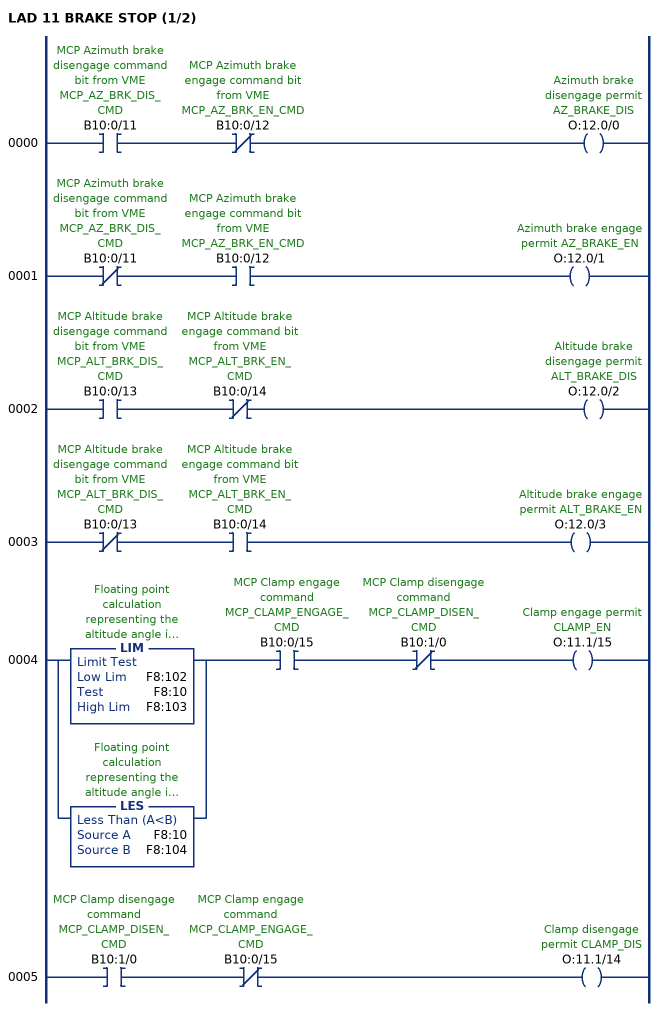
% Rung: 0 %
SOR XIC B10:0/11 XIO B10:0/12 OTE O:12.0/0 EOR
%   B10:0/11  MCP_AZ_BRK_DIS_CMD  "MCP Azimuth brake disengage command bit from VME" %
%   B10:0/12  MCP_AZ_BRK_EN_CMD  "MCP Azimuth brake engage command bit from VME" %
%   O:12.0/0  AZ_BRAKE_DIS  "Azimuth brake disengage permit" %
% Rung: 1 %
SOR XIO B10:0/11 XIC B10:0/12 OTE O:12.0/1 EOR
%   B10:0/11  MCP_AZ_BRK_DIS_CMD  "MCP Azimuth brake disengage command bit from VME" %
%   B10:0/12  MCP_AZ_BRK_EN_CMD  "MCP Azimuth brake engage command bit from VME" %
%   O:12.0/1  AZ_BRAKE_EN  "Azimuth brake engage permit" %
% Rung: 2 %
SOR XIC B10:0/13 XIO B10:0/14 OTE O:12.0/2 EOR
%   B10:0/13  MCP_ALT_BRK_DIS_CMD  "MCP Altitude brake disengage command bit from VME" %
%   B10:0/14  MCP_ALT_BRK_EN_CMD  "MCP Altitude brake engage command bit from VME" %
%   O:12.0/2  ALT_BRAKE_DIS  "Altitude brake disengage permit" %
% Rung: 3 %
SOR XIO B10:0/13 XIC B10:0/14 OTE O:12.0/3 EOR
%   B10:0/13  MCP_ALT_BRK_DIS_CMD  "MCP Altitude brake disengage command bit from VME" %
%   B10:0/14  MCP_ALT_BRK_EN_CMD  "MCP Altitude brake engage command bit from VME" %
%   O:12.0/3  ALT_BRAKE_EN  "Altitude brake engage permit" %
% Rung: 4 %
SOR BST LIM F8:102 F8:10 F8:103 NXB LES F8:10 F8:104 BND XIC B10:0/15 XIO B10:1/0 OTE O:11.1/15 EOR
%   F8:102  CLAMP_LOW_LIMIT  "The azimuth clamp will work above this limit and below CLAMP_HIGH_LIMIT" %
%   F8:10  ALT_ANGLE  "Floating point calculation representing the altitude angle in degrees." %
%   F8:103  CLAMP_HIGH_LIMIT  "The azimuth clamp will work below this limit and above CLAMP_LOW_LIMIT" %
%   F8:104  CLAMP_STOW_LIMIT  "The azimuth clamp will work below this limit" %
%   B10:0/15  MCP_CLAMP_ENGAGE_CMD  "MCP Clamp engage command" %
%   B10:1/0  MCP_CLAMP_DISEN_CMD  "MCP Clamp disengage command" %
%   O:11.1/15  CLAMP_EN  "Clamp engage permit" %
% Rung: 5 %
SOR XIC B10:1/0 XIO B10:0/15 OTE O:11.1/14 EOR
%   B10:1/0  MCP_CLAMP_DISEN_CMD  "MCP Clamp disengage command" %
%   B10:0/15  MCP_CLAMP_ENGAGE_CMD  "MCP Clamp engage command" %
%   O:11.1/14  CLAMP_DIS  "Clamp disengage permit" %

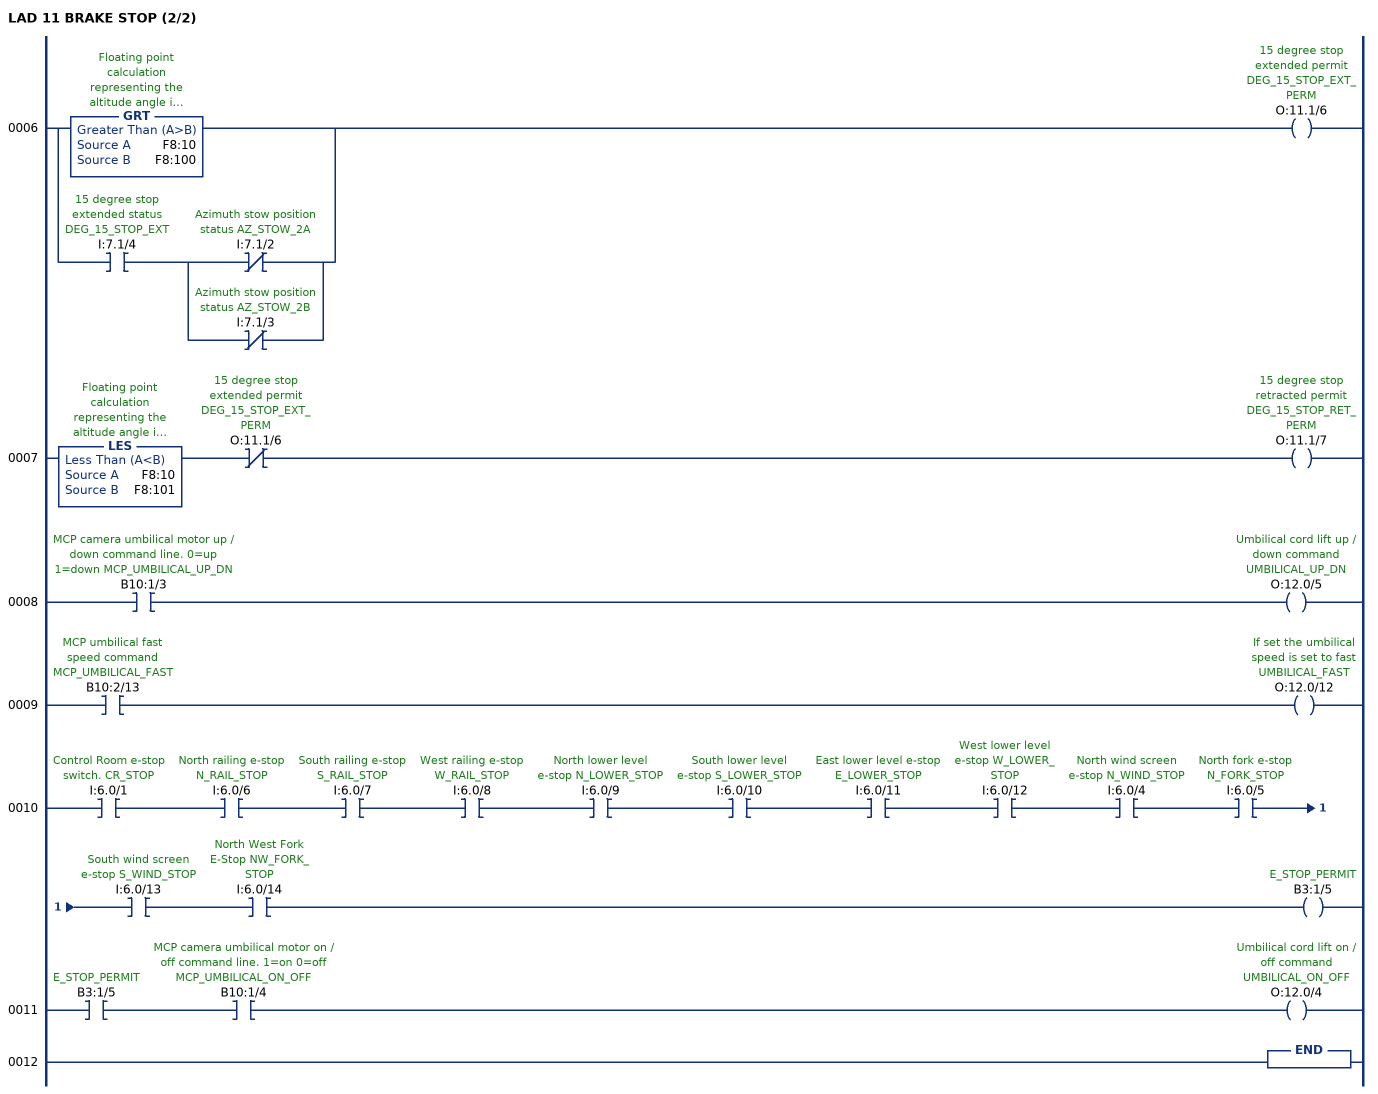
% Rung: 6 %
SOR BST GRT F8:10 F8:100 NXB XIC I:7.1/4 BST XIO I:7.1/2 NXB XIO I:7.1/3 BND BND OTE O:11.1/6 EOR
%   F8:10  ALT_ANGLE  "Floating point calculation representing the altitude angle in degrees." %
%   F8:100  DEG_15_STOP_EXT_LMT  "The 15 Degree stop extends at this value" %
%   I:7.1/4  DEG_15_STOP_EXT  "15 degree stop extended status" %
%   I:7.1/2  AZ_STOW_2A  "Azimuth stow position status" %
%   I:7.1/3  AZ_STOW_2B  "Azimuth stow position status" %
%   O:11.1/6  DEG_15_STOP_EXT_PERM  "15 degree stop extended permit" %
% Rung: 7 %
SOR LES F8:10 F8:101 XIO O:11.1/6 OTE O:11.1/7 EOR
%   F8:10  ALT_ANGLE  "Floating point calculation representing the altitude angle in degrees." %
%   F8:101  DEG_15_STOP_RET_LMT  "The 15 Degree stop retracts at this value" %
%   O:11.1/6  DEG_15_STOP_EXT_PERM  "15 degree stop extended permit" %
%   O:11.1/7  DEG_15_STOP_RET_PERM  "15 degree stop retracted permit" %
% Rung: 8 %
SOR XIC B10:1/3 OTE O:12.0/5 EOR
%   B10:1/3  MCP_UMBILICAL_UP_DN  "MCP camera umbilical motor up / down command line. 0=up 1=down" %
%   O:12.0/5  UMBILICAL_UP_DN  "Umbilical cord lift up / down command" %
% Rung: 9 %
SOR XIC B10:2/13 OTE O:12.0/12 EOR
%   B10:2/13  MCP_UMBILICAL_FAST  "MCP umbilical fast speed command" %
%   O:12.0/12  UMBILICAL_FAST  "If set the umbilical speed is set to fast" %
% Rung: 10 %
SOR XIC I:6.0/1 XIC I:6.0/6 XIC I:6.0/7 XIC I:6.0/8 XIC I:6.0/9 XIC I:6.0/10 XIC I:6.0/11 XIC I:6.0/12 XIC I:6.0/4 XIC I:6.0/5 XIC I:6.0/13 XIC I:6.0/14 OTE B3:1/5 EOR
%   I:6.0/1  CR_STOP  "Control Room e-stop switch." %
%   I:6.0/6  N_RAIL_STOP  "North railing e-stop" %
%   I:6.0/7  S_RAIL_STOP  "South railing e-stop" %
%   I:6.0/8  W_RAIL_STOP  "West railing e-stop" %
%   I:6.0/9  N_LOWER_STOP  "North lower level e-stop" %
%   I:6.0/10  S_LOWER_STOP  "South lower level e-stop" %
%   I:6.0/11  E_LOWER_STOP  "East lower level e-stop" %
%   I:6.0/12  W_LOWER_STOP  "West lower level e-stop" %
%   I:6.0/4  N_WIND_STOP  "North wind screen e-stop" %
%   I:6.0/5  N_FORK_STOP  "North fork e-stop" %
%   I:6.0/13  S_WIND_STOP  "South wind screen e-stop" %
%   I:6.0/14  NW_FORK_STOP  "North West Fork E-Stop" %
%   B3:1/5  E_STOP_PERMIT %
% Rung: 11 %
SOR XIC B3:1/5 XIC B10:1/4 OTE O:12.0/4 EOR
%   B3:1/5  E_STOP_PERMIT %
%   B10:1/4  MCP_UMBILICAL_ON_OFF  "MCP camera umbilical motor on / off command line. 1=on 0=off" %
%   O:12.0/4  UMBILICAL_ON_OFF  "Umbilical cord lift on / off command" %
% Rung: 12 %
SOR END EOR

LADDER 12 "E-STOP SW"
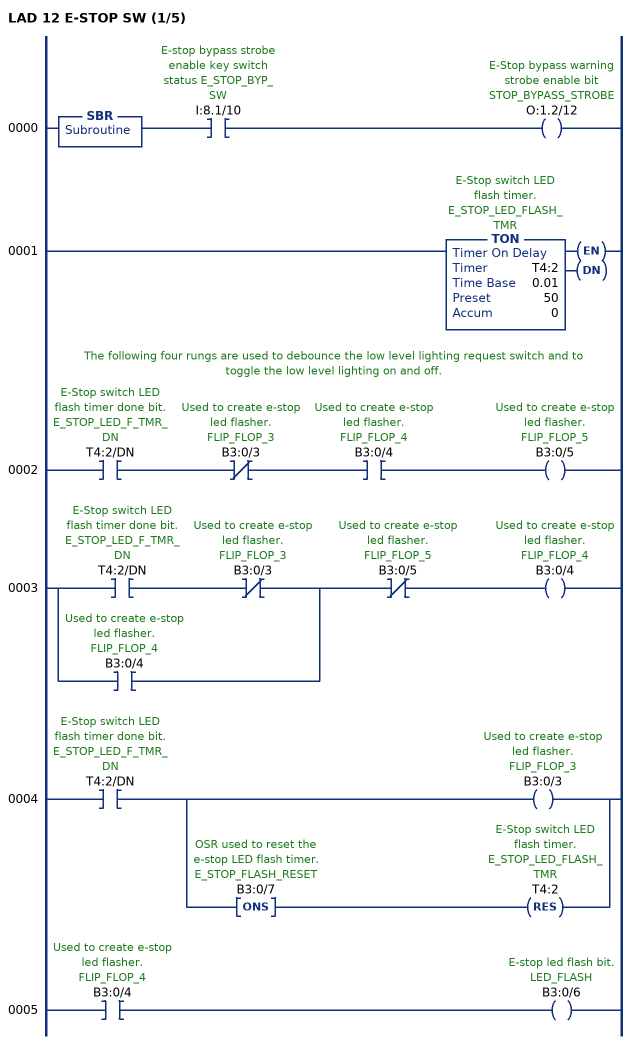
% Rung: 0 %
SOR SBR XIC I:8.1/10 OTE O:1.2/12 EOR
%   I:8.1/10  E_STOP_BYP_SW  "E-stop bypass strobe enable key switch status" %
%   O:1.2/12  STOP_BYPASS_STROBE  "E-Stop bypass warning strobe enable bit" %
% Rung: 1 %
SOR TON T4:2 0.01 50 0 EOR
%   T4:2  E_STOP_LED_FLASH_TMR  "E-Stop switch LED flash timer." %
% Rung: 2 %
% The following four rungs are used to debounce the low level lighting request switch and to toggle the low level lighting on and off. %
SOR XIC T4:2/DN XIO B3:0/3 XIC B3:0/4 OTE B3:0/5 EOR
%   T4:2/DN  E_STOP_LED_F_TMR_DN  "E-Stop switch LED flash timer done bit." %
%   B3:0/3  FLIP_FLOP_3  "Used to create e-stop led flasher." %
%   B3:0/4  FLIP_FLOP_4  "Used to create e-stop led flasher." %
%   B3:0/5  FLIP_FLOP_5  "Used to create e-stop led flasher." %
% Rung: 3 %
SOR BST XIC T4:2/DN XIO B3:0/3 NXB XIC B3:0/4 BND XIO B3:0/5 OTE B3:0/4 EOR
%   T4:2/DN  E_STOP_LED_F_TMR_DN  "E-Stop switch LED flash timer done bit." %
%   B3:0/3  FLIP_FLOP_3  "Used to create e-stop led flasher." %
%   B3:0/4  FLIP_FLOP_4  "Used to create e-stop led flasher." %
%   B3:0/5  FLIP_FLOP_5  "Used to create e-stop led flasher." %
% Rung: 4 %
SOR XIC T4:2/DN BST OTE B3:0/3 NXB OSR B3:0/7 RES T4:2 BND EOR
%   T4:2/DN  E_STOP_LED_F_TMR_DN  "E-Stop switch LED flash timer done bit." %
%   B3:0/3  FLIP_FLOP_3  "Used to create e-stop led flasher." %
%   B3:0/7  E_STOP_FLASH_RESET  "OSR used to reset the e-stop LED flash timer." %
%   T4:2  E_STOP_LED_FLASH_TMR  "E-Stop switch LED flash timer." %
% Rung: 5 %
SOR XIC B3:0/4 OTE B3:0/6 EOR
%   B3:0/4  FLIP_FLOP_4  "Used to create e-stop led flasher." %
%   B3:0/6  LED_FLASH  "E-stop led flash bit." %

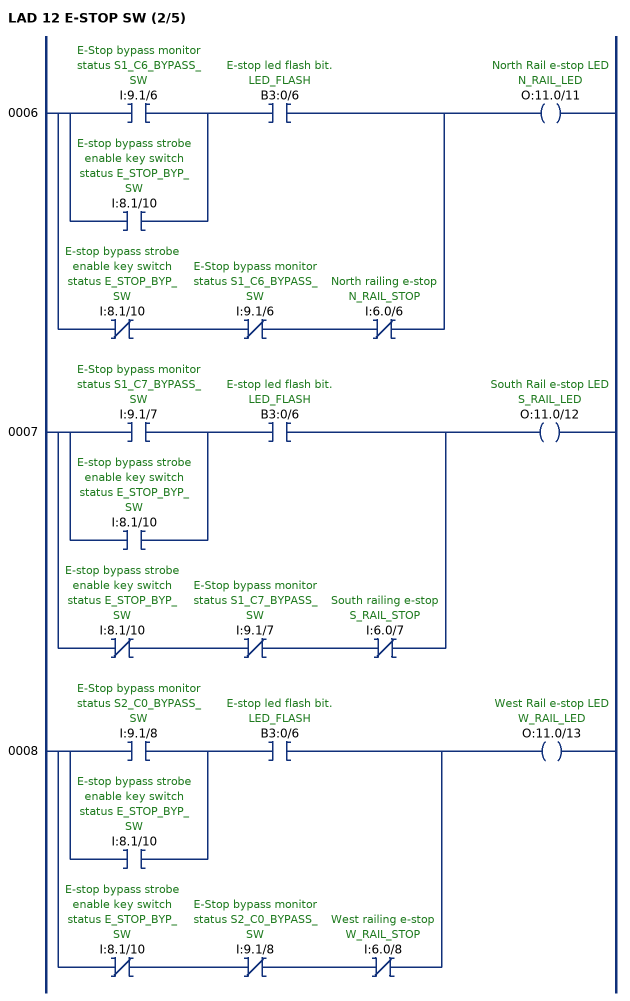
% Rung: 6 %
SOR BST BST XIC I:9.1/6 NXB XIC I:8.1/10 BND XIC B3:0/6 NXB XIO I:8.1/10 XIO I:9.1/6 XIO I:6.0/6 BND OTE O:11.0/11 EOR
%   I:9.1/6  S1_C6_BYPASS_SW  "E-Stop bypass monitor status" %
%   I:8.1/10  E_STOP_BYP_SW  "E-stop bypass strobe enable key switch status" %
%   B3:0/6  LED_FLASH  "E-stop led flash bit." %
%   I:6.0/6  N_RAIL_STOP  "North railing e-stop" %
%   O:11.0/11  N_RAIL_LED  "North Rail e-stop LED" %
% Rung: 7 %
SOR BST BST XIC I:9.1/7 NXB XIC I:8.1/10 BND XIC B3:0/6 NXB XIO I:8.1/10 XIO I:9.1/7 XIO I:6.0/7 BND OTE O:11.0/12 EOR
%   I:9.1/7  S1_C7_BYPASS_SW  "E-Stop bypass monitor status" %
%   I:8.1/10  E_STOP_BYP_SW  "E-stop bypass strobe enable key switch status" %
%   B3:0/6  LED_FLASH  "E-stop led flash bit." %
%   I:6.0/7  S_RAIL_STOP  "South railing e-stop" %
%   O:11.0/12  S_RAIL_LED  "South Rail e-stop LED" %
% Rung: 8 %
SOR BST BST XIC I:9.1/8 NXB XIC I:8.1/10 BND XIC B3:0/6 NXB XIO I:8.1/10 XIO I:9.1/8 XIO I:6.0/8 BND OTE O:11.0/13 EOR
%   I:9.1/8  S2_C0_BYPASS_SW  "E-Stop bypass monitor status" %
%   I:8.1/10  E_STOP_BYP_SW  "E-stop bypass strobe enable key switch status" %
%   B3:0/6  LED_FLASH  "E-stop led flash bit." %
%   I:6.0/8  W_RAIL_STOP  "West railing e-stop" %
%   O:11.0/13  W_RAIL_LED  "West Rail e-stop LED" %

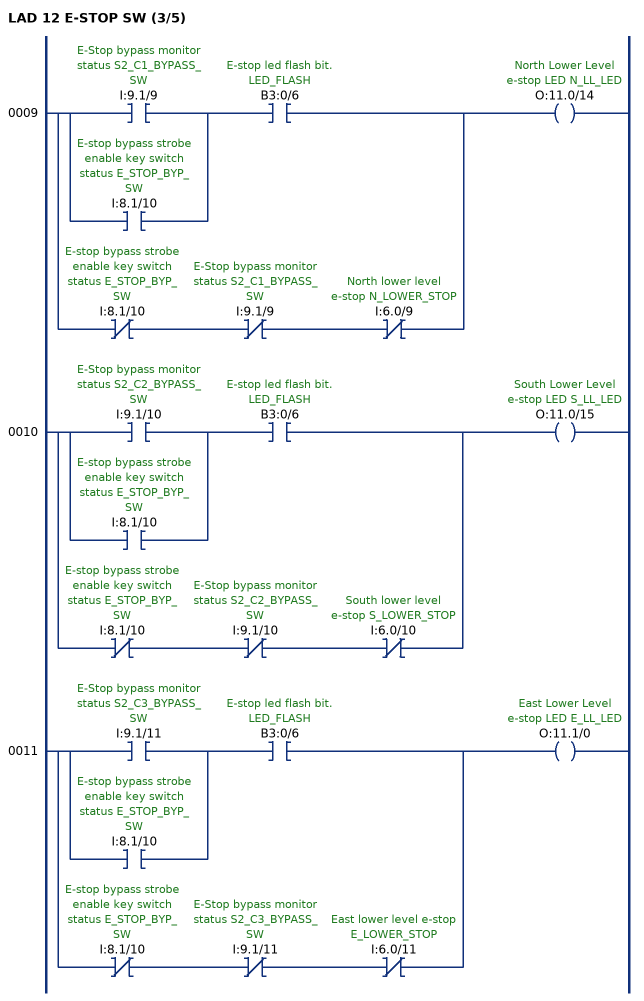
% Rung: 9 %
SOR BST BST XIC I:9.1/9 NXB XIC I:8.1/10 BND XIC B3:0/6 NXB XIO I:8.1/10 XIO I:9.1/9 XIO I:6.0/9 BND OTE O:11.0/14 EOR
%   I:9.1/9  S2_C1_BYPASS_SW  "E-Stop bypass monitor status" %
%   I:8.1/10  E_STOP_BYP_SW  "E-stop bypass strobe enable key switch status" %
%   B3:0/6  LED_FLASH  "E-stop led flash bit." %
%   I:6.0/9  N_LOWER_STOP  "North lower level e-stop" %
%   O:11.0/14  N_LL_LED  "North Lower Level e-stop LED" %
% Rung: 10 %
SOR BST BST XIC I:9.1/10 NXB XIC I:8.1/10 BND XIC B3:0/6 NXB XIO I:8.1/10 XIO I:9.1/10 XIO I:6.0/10 BND OTE O:11.0/15 EOR
%   I:9.1/10  S2_C2_BYPASS_SW  "E-Stop bypass monitor status" %
%   I:8.1/10  E_STOP_BYP_SW  "E-stop bypass strobe enable key switch status" %
%   B3:0/6  LED_FLASH  "E-stop led flash bit." %
%   I:6.0/10  S_LOWER_STOP  "South lower level e-stop" %
%   O:11.0/15  S_LL_LED  "South Lower Level e-stop LED" %
% Rung: 11 %
SOR BST BST XIC I:9.1/11 NXB XIC I:8.1/10 BND XIC B3:0/6 NXB XIO I:8.1/10 XIO I:9.1/11 XIO I:6.0/11 BND OTE O:11.1/0 EOR
%   I:9.1/11  S2_C3_BYPASS_SW  "E-Stop bypass monitor status" %
%   I:8.1/10  E_STOP_BYP_SW  "E-stop bypass strobe enable key switch status" %
%   B3:0/6  LED_FLASH  "E-stop led flash bit." %
%   I:6.0/11  E_LOWER_STOP  "East lower level e-stop" %
%   O:11.1/0  E_LL_LED  "East Lower Level e-stop LED" %

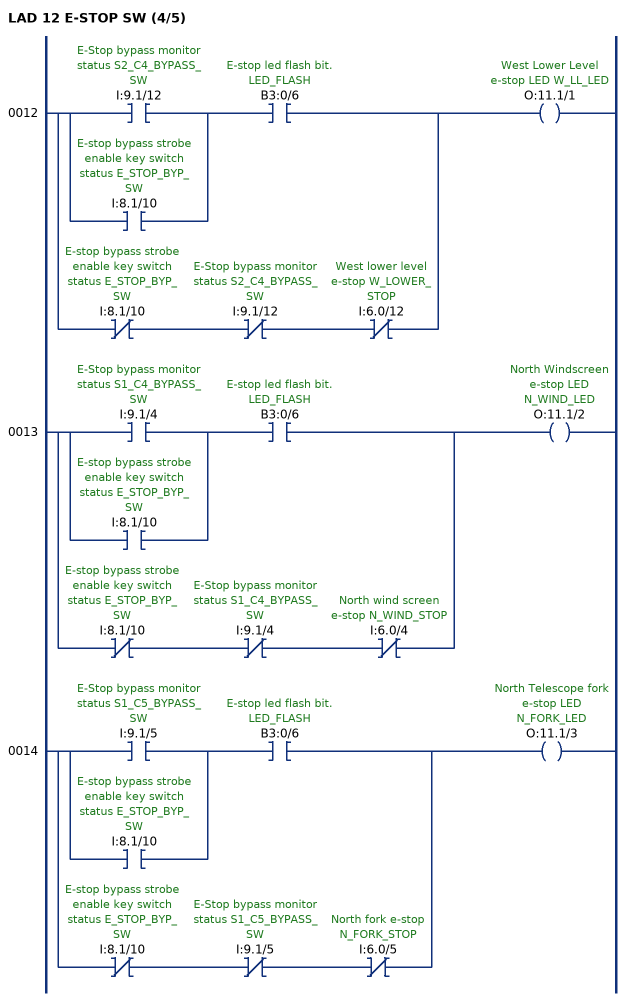
% Rung: 12 %
SOR BST BST XIC I:9.1/12 NXB XIC I:8.1/10 BND XIC B3:0/6 NXB XIO I:8.1/10 XIO I:9.1/12 XIO I:6.0/12 BND OTE O:11.1/1 EOR
%   I:9.1/12  S2_C4_BYPASS_SW  "E-Stop bypass monitor status" %
%   I:8.1/10  E_STOP_BYP_SW  "E-stop bypass strobe enable key switch status" %
%   B3:0/6  LED_FLASH  "E-stop led flash bit." %
%   I:6.0/12  W_LOWER_STOP  "West lower level e-stop" %
%   O:11.1/1  W_LL_LED  "West Lower Level e-stop LED" %
% Rung: 13 %
SOR BST BST XIC I:9.1/4 NXB XIC I:8.1/10 BND XIC B3:0/6 NXB XIO I:8.1/10 XIO I:9.1/4 XIO I:6.0/4 BND OTE O:11.1/2 EOR
%   I:9.1/4  S1_C4_BYPASS_SW  "E-Stop bypass monitor status" %
%   I:8.1/10  E_STOP_BYP_SW  "E-stop bypass strobe enable key switch status" %
%   B3:0/6  LED_FLASH  "E-stop led flash bit." %
%   I:6.0/4  N_WIND_STOP  "North wind screen e-stop" %
%   O:11.1/2  N_WIND_LED  "North Windscreen e-stop LED" %
% Rung: 14 %
SOR BST BST XIC I:9.1/5 NXB XIC I:8.1/10 BND XIC B3:0/6 NXB XIO I:8.1/10 XIO I:9.1/5 XIO I:6.0/5 BND OTE O:11.1/3 EOR
%   I:9.1/5  S1_C5_BYPASS_SW  "E-Stop bypass monitor status" %
%   I:8.1/10  E_STOP_BYP_SW  "E-stop bypass strobe enable key switch status" %
%   B3:0/6  LED_FLASH  "E-stop led flash bit." %
%   I:6.0/5  N_FORK_STOP  "North fork e-stop" %
%   O:11.1/3  N_FORK_LED  "North Telescope fork e-stop LED" %

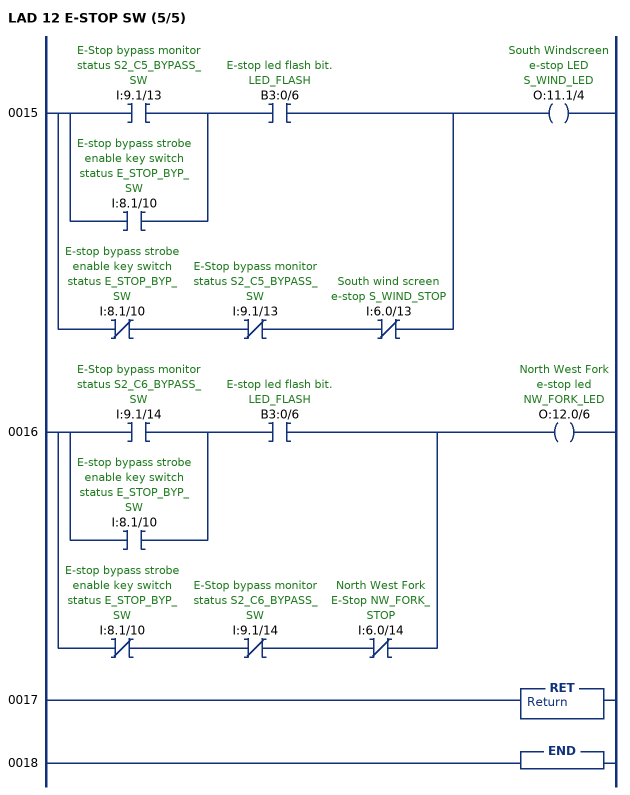
% Rung: 15 %
SOR BST BST XIC I:9.1/13 NXB XIC I:8.1/10 BND XIC B3:0/6 NXB XIO I:8.1/10 XIO I:9.1/13 XIO I:6.0/13 BND OTE O:11.1/4 EOR
%   I:9.1/13  S2_C5_BYPASS_SW  "E-Stop bypass monitor status" %
%   I:8.1/10  E_STOP_BYP_SW  "E-stop bypass strobe enable key switch status" %
%   B3:0/6  LED_FLASH  "E-stop led flash bit." %
%   I:6.0/13  S_WIND_STOP  "South wind screen e-stop" %
%   O:11.1/4  S_WIND_LED  "South Windscreen e-stop LED" %
% Rung: 16 %
SOR BST BST XIC I:9.1/14 NXB XIC I:8.1/10 BND XIC B3:0/6 NXB XIO I:8.1/10 XIO I:9.1/14 XIO I:6.0/14 BND OTE O:12.0/6 EOR
%   I:9.1/14  S2_C6_BYPASS_SW  "E-Stop bypass monitor status" %
%   I:8.1/10  E_STOP_BYP_SW  "E-stop bypass strobe enable key switch status" %
%   B3:0/6  LED_FLASH  "E-stop led flash bit." %
%   I:6.0/14  NW_FORK_STOP  "North West Fork E-Stop" %
%   O:12.0/6  NW_FORK_LED  "North West Fork e-stop led" %
% Rung: 17 %
SOR RET EOR
% Rung: 18 %
SOR END EOR

LADDER 13 "SPEC CONT"    % Spectrograph Controls %
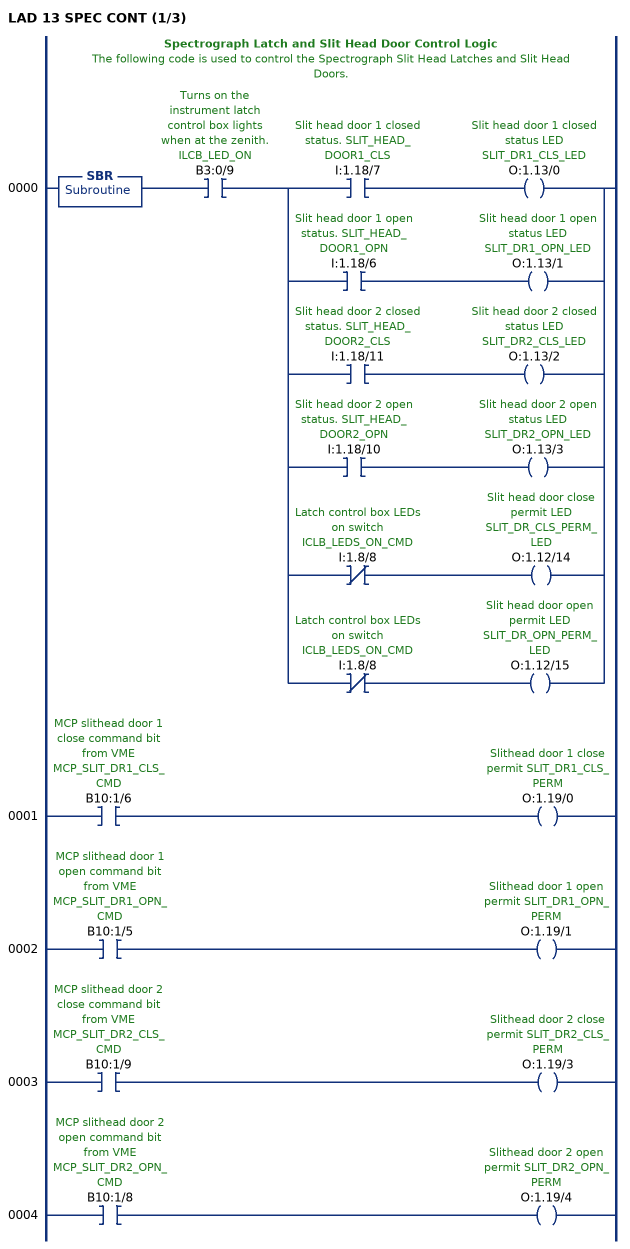
% Rung: 0 %
% TITLE: Spectrograph Latch and Slit Head Door Control Logic %
% The following code is used to control the Spectrograph Slit Head Latches and Slit Head Doors. %
SOR SBR XIC B3:0/9 BST XIC I:1.18/7 OTE O:1.13/0 NXB XIC I:1.18/6 OTE O:1.13/1 NXB XIC I:1.18/11 OTE O:1.13/2 NXB XIC I:1.18/10 OTE O:1.13/3 NXB XIO I:1.8/8 OTE O:1.12/14 NXB XIO I:1.8/8 OTE O:1.12/15 BND EOR
%   B3:0/9  ILCB_LED_ON  "Turns on the instrument latch control box lights when at the zenith." %
%   I:1.18/7  SLIT_HEAD_DOOR1_CLS  "Slit head door 1 closed status." %
%   O:1.13/0  SLIT_DR1_CLS_LED  "Slit head door 1 closed status LED" %
%   I:1.18/6  SLIT_HEAD_DOOR1_OPN  "Slit head door 1 open status." %
%   O:1.13/1  SLIT_DR1_OPN_LED  "Slit head door 1 open status LED" %
%   I:1.18/11  SLIT_HEAD_DOOR2_CLS  "Slit head door 2 closed status." %
%   O:1.13/2  SLIT_DR2_CLS_LED  "Slit head door 2 closed status LED" %
%   I:1.18/10  SLIT_HEAD_DOOR2_OPN  "Slit head door 2 open status." %
%   O:1.13/3  SLIT_DR2_OPN_LED  "Slit head door 2 open status LED" %
%   I:1.8/8  ICLB_LEDS_ON_CMD  "Latch control box LEDs on switch" %
%   O:1.12/14  SLIT_DR_CLS_PERM_LED  "Slit head door close permit LED" %
%   O:1.12/15  SLIT_DR_OPN_PERM_LED  "Slit head door open permit LED" %
% Rung: 1 %
SOR XIC B10:1/6 OTE O:1.19/0 EOR
%   B10:1/6  MCP_SLIT_DR1_CLS_CMD  "MCP slithead door 1 close command bit from VME" %
%   O:1.19/0  SLIT_DR1_CLS_PERM  "Slithead door 1 close permit" %
% Rung: 2 %
SOR XIC B10:1/5 OTE O:1.19/1 EOR
%   B10:1/5  MCP_SLIT_DR1_OPN_CMD  "MCP slithead door 1 open command bit from VME" %
%   O:1.19/1  SLIT_DR1_OPN_PERM  "Slithead door 1 open permit" %
% Rung: 3 %
SOR XIC B10:1/9 OTE O:1.19/3 EOR
%   B10:1/9  MCP_SLIT_DR2_CLS_CMD  "MCP slithead door 2 close command bit from VME" %
%   O:1.19/3  SLIT_DR2_CLS_PERM  "Slithead door 2 close permit" %
% Rung: 4 %
SOR XIC B10:1/8 OTE O:1.19/4 EOR
%   B10:1/8  MCP_SLIT_DR2_OPN_CMD  "MCP slithead door 2 open command bit from VME" %
%   O:1.19/4  SLIT_DR2_OPN_PERM  "Slithead door 2 open permit" %

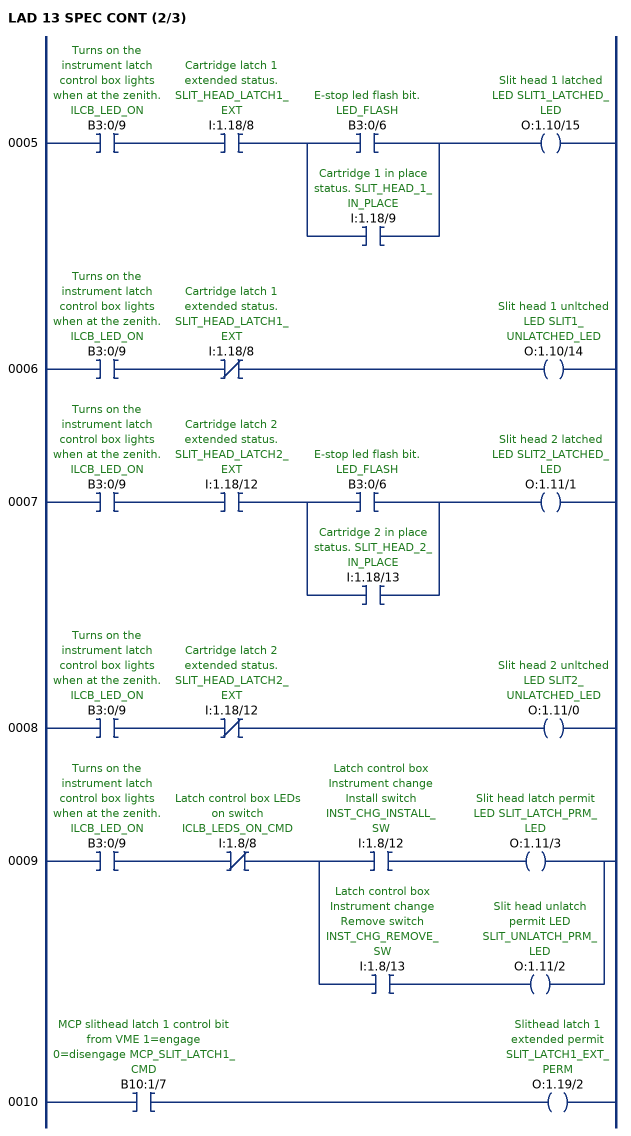
% Rung: 5 %
SOR XIC B3:0/9 XIC I:1.18/8 BST XIC B3:0/6 NXB XIC I:1.18/9 BND OTE O:1.10/15 EOR
%   B3:0/9  ILCB_LED_ON  "Turns on the instrument latch control box lights when at the zenith." %
%   I:1.18/8  SLIT_HEAD_LATCH1_EXT  "Cartridge latch 1 extended status." %
%   B3:0/6  LED_FLASH  "E-stop led flash bit." %
%   I:1.18/9  SLIT_HEAD_1_IN_PLACE  "Cartridge 1 in place status." %
%   O:1.10/15  SLIT1_LATCHED_LED  "Slit head 1 latched LED" %
% Rung: 6 %
SOR XIC B3:0/9 XIO I:1.18/8 OTE O:1.10/14 EOR
%   B3:0/9  ILCB_LED_ON  "Turns on the instrument latch control box lights when at the zenith." %
%   I:1.18/8  SLIT_HEAD_LATCH1_EXT  "Cartridge latch 1 extended status." %
%   O:1.10/14  SLIT1_UNLATCHED_LED  "Slit head 1 unltched LED" %
% Rung: 7 %
SOR XIC B3:0/9 XIC I:1.18/12 BST XIC B3:0/6 NXB XIC I:1.18/13 BND OTE O:1.11/1 EOR
%   B3:0/9  ILCB_LED_ON  "Turns on the instrument latch control box lights when at the zenith." %
%   I:1.18/12  SLIT_HEAD_LATCH2_EXT  "Cartridge latch 2 extended status." %
%   B3:0/6  LED_FLASH  "E-stop led flash bit." %
%   I:1.18/13  SLIT_HEAD_2_IN_PLACE  "Cartridge 2 in place status." %
%   O:1.11/1  SLIT2_LATCHED_LED  "Slit head 2 latched LED" %
% Rung: 8 %
SOR XIC B3:0/9 XIO I:1.18/12 OTE O:1.11/0 EOR
%   B3:0/9  ILCB_LED_ON  "Turns on the instrument latch control box lights when at the zenith." %
%   I:1.18/12  SLIT_HEAD_LATCH2_EXT  "Cartridge latch 2 extended status." %
%   O:1.11/0  SLIT2_UNLATCHED_LED  "Slit head 2 unltched LED" %
% Rung: 9 %
SOR XIC B3:0/9 XIO I:1.8/8 BST XIC I:1.8/12 OTE O:1.11/3 NXB XIC I:1.8/13 OTE O:1.11/2 BND EOR
%   B3:0/9  ILCB_LED_ON  "Turns on the instrument latch control box lights when at the zenith." %
%   I:1.8/8  ICLB_LEDS_ON_CMD  "Latch control box LEDs on switch" %
%   I:1.8/12  INST_CHG_INSTALL_SW  "Latch control box Instrument change Install switch" %
%   O:1.11/3  SLIT_LATCH_PRM_LED  "Slit head latch permit LED" %
%   I:1.8/13  INST_CHG_REMOVE_SW  "Latch control box Instrument change Remove switch" %
%   O:1.11/2  SLIT_UNLATCH_PRM_LED  "Slit head unlatch permit LED" %
% Rung: 10 %
SOR XIC B10:1/7 OTE O:1.19/2 EOR
%   B10:1/7  MCP_SLIT_LATCH1_CMD  "MCP slithead latch 1 control bit from VME 1=engage 0=disengage" %
%   O:1.19/2  SLIT_LATCH1_EXT_PERM  "Slithead latch 1 extended permit" %

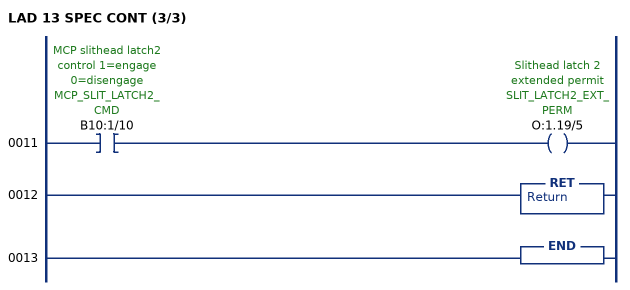
% Rung: 11 %
SOR XIC B10:1/10 OTE O:1.19/5 EOR
%   B10:1/10  MCP_SLIT_LATCH2_CMD  "MCP slithead latch2 control 1=engage 0=disengage" %
%   O:1.19/5  SLIT_LATCH2_EXT_PERM  "Slithead latch 2 extended permit" %
% Rung: 12 %
SOR RET EOR
% Rung: 13 %
SOR END EOR

LADDER 14 "FLAT FIELD"    % Flat Field Lamp Controls %
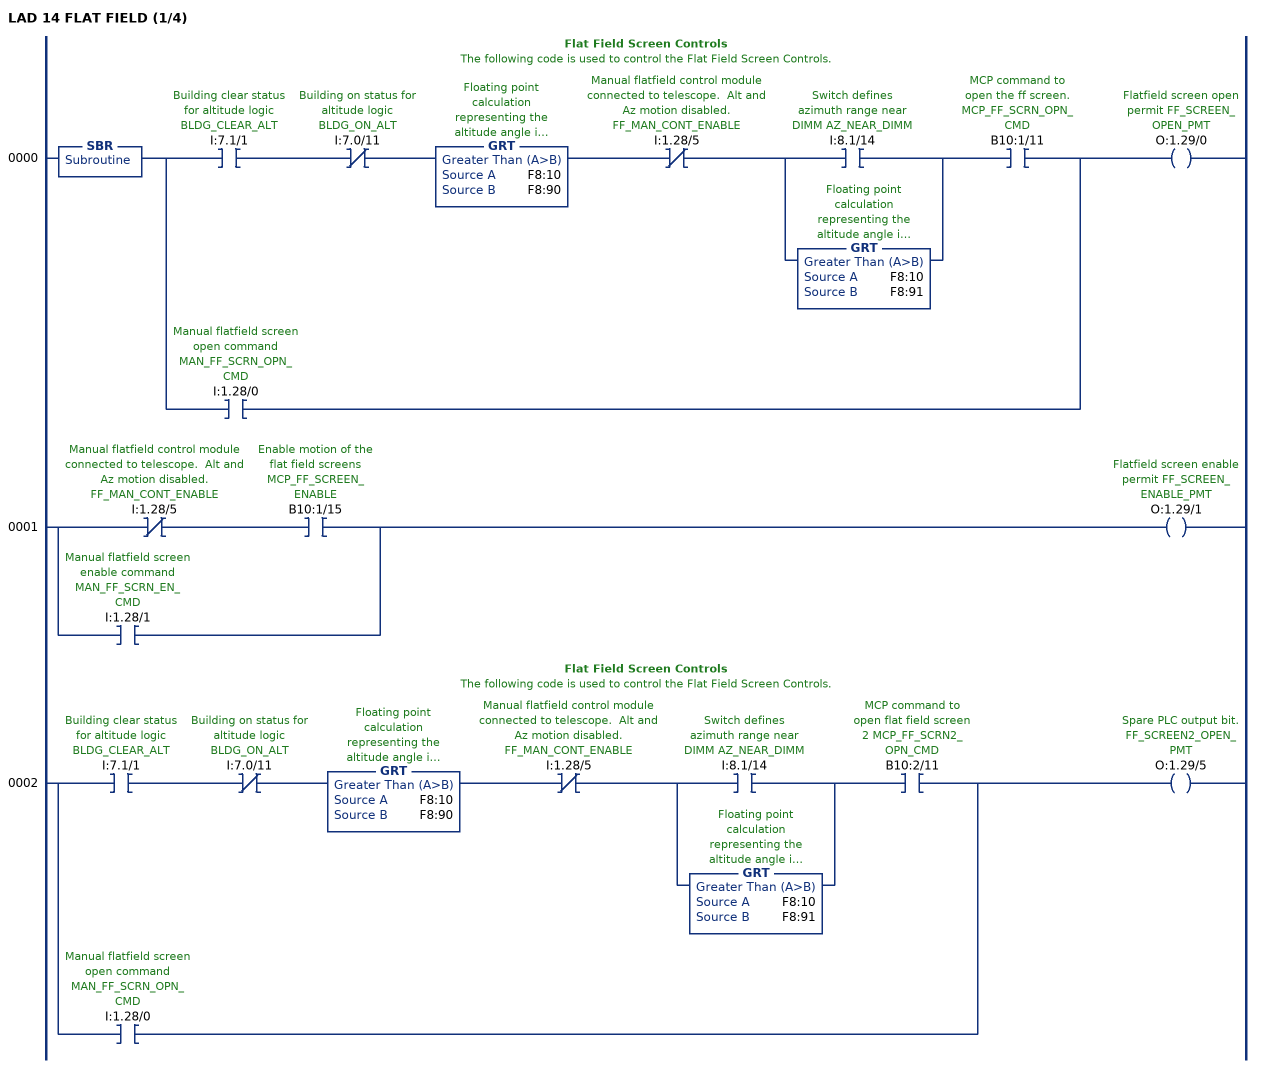
% Rung: 0 %
% TITLE: Flat Field Screen Controls %
% The following code is used to control the Flat Field Screen Controls. %
SOR SBR BST XIC I:7.1/1 XIO I:7.0/11 GRT F8:10 F8:90 XIO I:1.28/5 BST XIC I:8.1/14 NXB GRT F8:10 F8:91 BND XIC B10:1/11 NXB XIC I:1.28/0 BND OTE O:1.29/0 EOR
%   I:7.1/1  BLDG_CLEAR_ALT  "Building clear status for altitude logic" %
%   I:7.0/11  BLDG_ON_ALT  "Building on status for altitude logic" %
%   F8:10  ALT_ANGLE  "Floating point calculation representing the altitude angle in degrees." %
%   F8:90  FF_SCREEN_ALT_LIMIT  "Flatfield screen altitude limit" %
%   I:1.28/5  FF_MAN_CONT_ENABLE  "Manual flatfield control module connected to telescope.  Alt and Az motion disabled." %
%   I:8.1/14  AZ_NEAR_DIMM  "Switch defines azimuth range near DIMM" %
%   F8:91  FFS_DIMM_ALT_LIM  "Lower Altitude Limit for FFS Enable In DIMM Avoidance Zone" %
%   B10:1/11  MCP_FF_SCRN_OPN_CMD  "MCP command to open the ff screen." %
%   I:1.28/0  MAN_FF_SCRN_OPN_CMD  "Manual flatfield screen open command" %
%   O:1.29/0  FF_SCREEN_OPEN_PMT  "Flatfield screen open permit" %
% Rung: 1 %
SOR BST XIO I:1.28/5 XIC B10:1/15 NXB XIC I:1.28/1 BND OTE O:1.29/1 EOR
%   I:1.28/5  FF_MAN_CONT_ENABLE  "Manual flatfield control module connected to telescope.  Alt and Az motion disabled." %
%   B10:1/15  MCP_FF_SCREEN_ENABLE  "Enable motion of the flat field screens" %
%   I:1.28/1  MAN_FF_SCRN_EN_CMD  "Manual flatfield screen enable command" %
%   O:1.29/1  FF_SCREEN_ENABLE_PMT  "Flatfield screen enable permit" %
% Rung: 2 %
% TITLE: Flat Field Screen Controls %
% The following code is used to control the Flat Field Screen Controls. %
SOR BST XIC I:7.1/1 XIO I:7.0/11 GRT F8:10 F8:90 XIO I:1.28/5 BST XIC I:8.1/14 NXB GRT F8:10 F8:91 BND XIC B10:2/11 NXB XIC I:1.28/0 BND OTE O:1.29/5 EOR
%   I:7.1/1  BLDG_CLEAR_ALT  "Building clear status for altitude logic" %
%   I:7.0/11  BLDG_ON_ALT  "Building on status for altitude logic" %
%   F8:10  ALT_ANGLE  "Floating point calculation representing the altitude angle in degrees." %
%   F8:90  FF_SCREEN_ALT_LIMIT  "Flatfield screen altitude limit" %
%   I:1.28/5  FF_MAN_CONT_ENABLE  "Manual flatfield control module connected to telescope.  Alt and Az motion disabled." %
%   I:8.1/14  AZ_NEAR_DIMM  "Switch defines azimuth range near DIMM" %
%   F8:91  FFS_DIMM_ALT_LIM  "Lower Altitude Limit for FFS Enable In DIMM Avoidance Zone" %
%   B10:2/11  MCP_FF_SCRN2_OPN_CMD  "MCP command to open flat field screen 2" %
%   I:1.28/0  MAN_FF_SCRN_OPN_CMD  "Manual flatfield screen open command" %
%   O:1.29/5  FF_SCREEN2_OPEN_PMT  "Spare PLC output bit." %

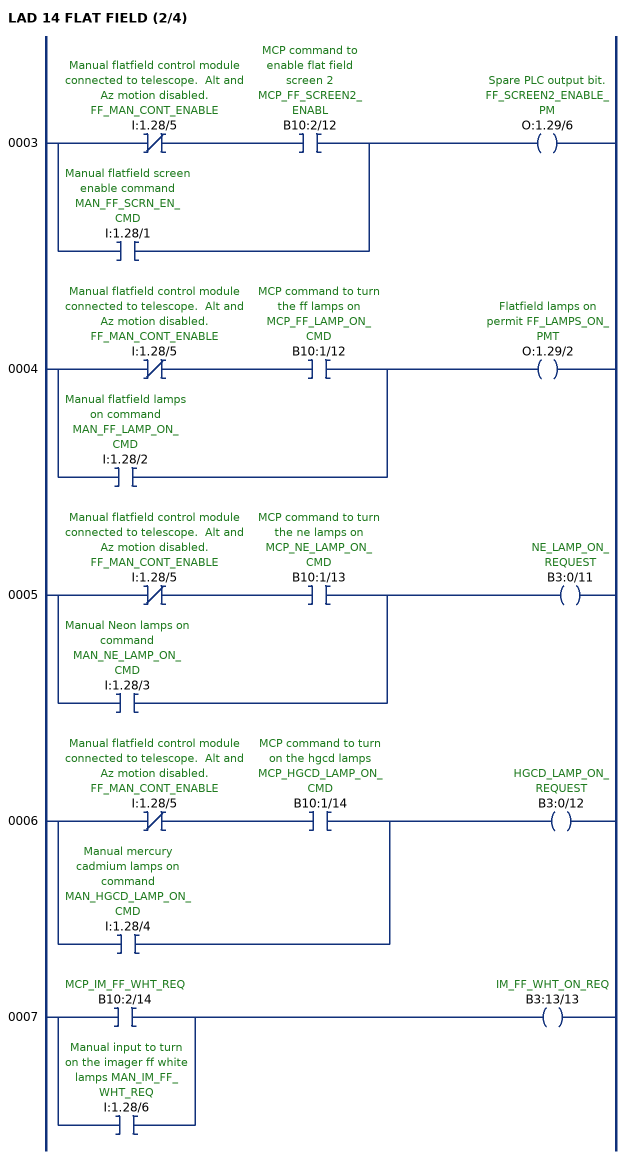
% Rung: 3 %
SOR BST XIO I:1.28/5 XIC B10:2/12 NXB XIC I:1.28/1 BND OTE O:1.29/6 EOR
%   I:1.28/5  FF_MAN_CONT_ENABLE  "Manual flatfield control module connected to telescope.  Alt and Az motion disabled." %
%   B10:2/12  MCP_FF_SCREEN2_ENABL  "MCP command to enable flat field screen 2" %
%   I:1.28/1  MAN_FF_SCRN_EN_CMD  "Manual flatfield screen enable command" %
%   O:1.29/6  FF_SCREEN2_ENABLE_PM  "Spare PLC output bit." %
% Rung: 4 %
SOR BST XIO I:1.28/5 XIC B10:1/12 NXB XIC I:1.28/2 BND OTE O:1.29/2 EOR
%   I:1.28/5  FF_MAN_CONT_ENABLE  "Manual flatfield control module connected to telescope.  Alt and Az motion disabled." %
%   B10:1/12  MCP_FF_LAMP_ON_CMD  "MCP command to turn the ff lamps on" %
%   I:1.28/2  MAN_FF_LAMP_ON_CMD  "Manual flatfield lamps on command" %
%   O:1.29/2  FF_LAMPS_ON_PMT  "Flatfield lamps on permit" %
% Rung: 5 %
SOR BST XIO I:1.28/5 XIC B10:1/13 NXB XIC I:1.28/3 BND OTE B3:0/11 EOR
%   I:1.28/5  FF_MAN_CONT_ENABLE  "Manual flatfield control module connected to telescope.  Alt and Az motion disabled." %
%   B10:1/13  MCP_NE_LAMP_ON_CMD  "MCP command to turn the ne lamps on" %
%   I:1.28/3  MAN_NE_LAMP_ON_CMD  "Manual Neon lamps on command" %
%   B3:0/11  NE_LAMP_ON_REQUEST %
% Rung: 6 %
SOR BST XIO I:1.28/5 XIC B10:1/14 NXB XIC I:1.28/4 BND OTE B3:0/12 EOR
%   I:1.28/5  FF_MAN_CONT_ENABLE  "Manual flatfield control module connected to telescope.  Alt and Az motion disabled." %
%   B10:1/14  MCP_HGCD_LAMP_ON_CMD  "MCP command to turn on the hgcd lamps" %
%   I:1.28/4  MAN_HGCD_LAMP_ON_CMD  "Manual mercury cadmium lamps on command" %
%   B3:0/12  HGCD_LAMP_ON_REQUEST %
% Rung: 7 %
SOR BST XIC B10:2/14 NXB XIC I:1.28/6 BND OTE B3:13/13 EOR
%   B10:2/14  MCP_IM_FF_WHT_REQ %
%   I:1.28/6  MAN_IM_FF_WHT_REQ  "Manual input to turn on the imager ff white lamps" %
%   B3:13/13  IM_FF_WHT_ON_REQ %

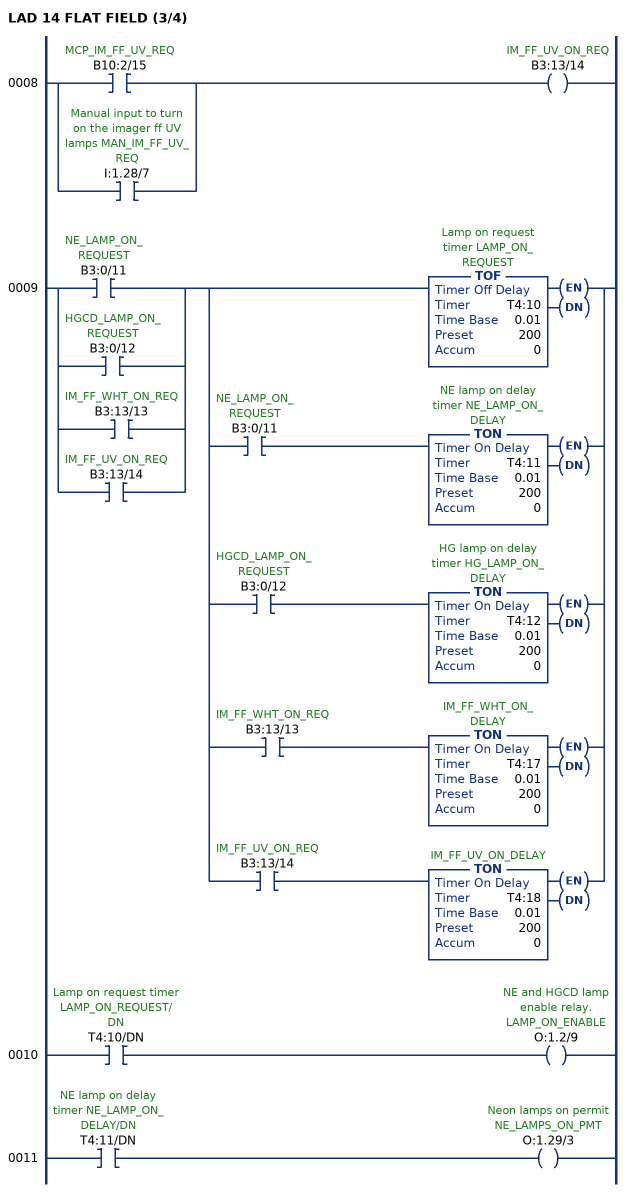
% Rung: 8 %
SOR BST XIC B10:2/15 NXB XIC I:1.28/7 BND OTE B3:13/14 EOR
%   B10:2/15  MCP_IM_FF_UV_REQ %
%   I:1.28/7  MAN_IM_FF_UV_REQ  "Manual input to turn on the imager ff UV lamps" %
%   B3:13/14  IM_FF_UV_ON_REQ %
% Rung: 9 %
SOR BST XIC B3:0/11 NXB XIC B3:0/12 NXB XIC B3:13/13 NXB XIC B3:13/14 BND BST TOF T4:10 0.01 200 0 NXB XIC B3:0/11 TON T4:11 0.01 200 0 NXB XIC B3:0/12 TON T4:12 0.01 200 0 NXB XIC B3:13/13 TON T4:17 0.01 200 0 NXB XIC B3:13/14 TON T4:18 0.01 200 0 BND EOR
%   B3:0/11  NE_LAMP_ON_REQUEST %
%   B3:0/12  HGCD_LAMP_ON_REQUEST %
%   B3:13/13  IM_FF_WHT_ON_REQ %
%   B3:13/14  IM_FF_UV_ON_REQ %
%   T4:10  LAMP_ON_REQUEST  "Lamp on request timer" %
%   T4:11  NE_LAMP_ON_DELAY  "NE lamp on delay timer" %
%   T4:12  HG_LAMP_ON_DELAY  "HG lamp on delay timer" %
%   T4:17  IM_FF_WHT_ON_DELAY %
%   T4:18  IM_FF_UV_ON_DELAY %
% Rung: 10 %
SOR XIC T4:10/DN OTE O:1.2/9 EOR
%   T4:10  LAMP_ON_REQUEST  "Lamp on request timer" %
%   O:1.2/9  LAMP_ON_ENABLE  "NE and HGCD lamp enable relay." %
% Rung: 11 %
SOR XIC T4:11/DN OTE O:1.29/3 EOR
%   T4:11  NE_LAMP_ON_DELAY  "NE lamp on delay timer" %
%   O:1.29/3  NE_LAMPS_ON_PMT  "Neon lamps on permit" %

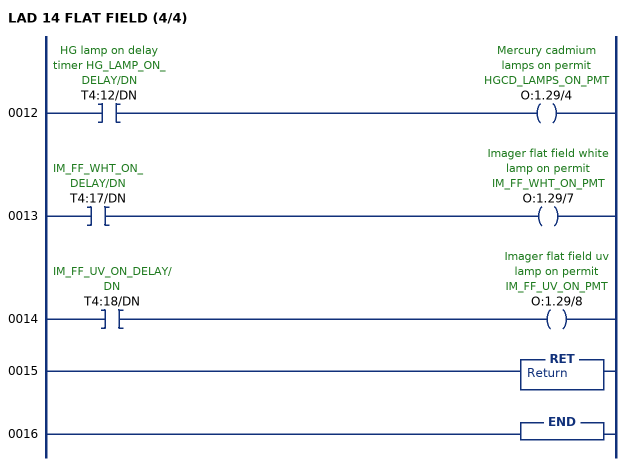
% Rung: 12 %
SOR XIC T4:12/DN OTE O:1.29/4 EOR
%   T4:12  HG_LAMP_ON_DELAY  "HG lamp on delay timer" %
%   O:1.29/4  HGCD_LAMPS_ON_PMT  "Mercury cadmium lamps on permit" %
% Rung: 13 %
SOR XIC T4:17/DN OTE O:1.29/7 EOR
%   T4:17  IM_FF_WHT_ON_DELAY %
%   O:1.29/7  IM_FF_WHT_ON_PMT  "Imager flat field white lamp on permit" %
% Rung: 14 %
SOR XIC T4:18/DN OTE O:1.29/8 EOR
%   T4:18  IM_FF_UV_ON_DELAY %
%   O:1.29/8  IM_FF_UV_ON_PMT  "Imager flat field uv lamp on permit" %
% Rung: 15 %
SOR RET EOR
% Rung: 16 %
SOR END EOR

LADDER 15 "FLEXANALOG"    % Flex I/O Analog Routines %
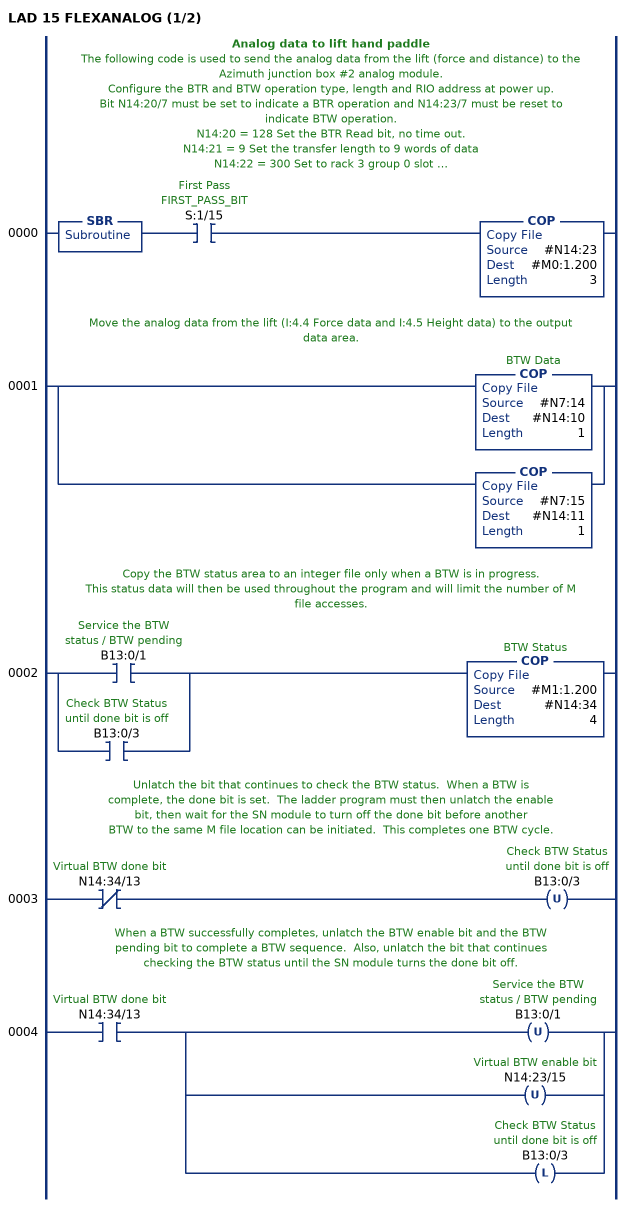
% Rung: 0 %
% TITLE: Analog data to lift hand paddle %
% The following code is used to send the analog data from the lift (force and distance) to the Azimuth junction box #2 analog module.
% 
% Configure the BTR and BTW operation type, length and RIO address at power up.
% Bit N14:20/7 must be set to indicate a BTR operation and N14:23/7 must be reset to indicate BTW operation.
% 
% N14:20 = 128 Set the BTR Read bit, no time out.
% N14:21 = 9 Set the transfer length to 9 words of data
% N14:22 = 300 Set to rack 3 group 0 slot 0
% 
% N14:23 = 0 Set the BTW write  bit, no time out.
% N14:24 = 1 Set the transfer length to 8 word of data
% N14:25 = 300 Set to rack 3 group 0 slot 0 %
SOR SBR XIC S:1/15 COP #N14:23 #M0:1.200 3 EOR
%   S:1/15  FIRST_PASS_BIT  "First Pass" %
% Rung: 1 %
% Move the analog data from the lift (I:4.4 Force data and I:4.5 Height data) to the output data area. %
SOR BST COP #N7:14 #N14:10 1 NXB COP #N7:15 #N14:11 1 BND EOR
%   N7:14  LIFT_FORCE_DISPLAY  "Instrument lift hand held force display scale factors." %
%   N14:10  "BTW Data" %
%   N7:15  LIFT_DIST_DISPLAY  "Instrument lift hand held distance display scale factors." %
% Rung: 2 %
% Copy the BTW status area to an integer file only when a BTW is in progress.
% This status data will then be used throughout the program and will limit the number of M file accesses. %
SOR BST XIC B13:0/1 NXB XIC B13:0/3 BND COP #M1:1.200 #N14:34 4 EOR
%   B13:0/1  "Service the BTW status / BTW pending" %
%   B13:0/3  "Check BTW Status until done bit is off" %
%   N14:34  "BTW Status" %
% Rung: 3 %
% Unlatch the bit that continues to check the BTW status.  When a BTW is
% complete, the done bit is set.  The ladder program must then unlatch the enable
% bit, then wait for the SN module to turn off the done bit before another
% BTW to the same M file location can be initiated.  This completes one BTW cycle. %
SOR XIO N14:34/13 OTU B13:0/3 EOR
%   N14:34/13  "Virtual BTW done bit" %
%   B13:0/3  "Check BTW Status until done bit is off" %
% Rung: 4 %
% When a BTW successfully completes, unlatch the BTW enable bit and the BTW
% pending bit to complete a BTW sequence.  Also, unlatch the bit that continues
% checking the BTW status until the SN module turns the done bit off. %
SOR XIC N14:34/13 BST OTU B13:0/1 NXB OTU N14:23/15 NXB OTL B13:0/3 BND EOR
%   N14:34/13  "Virtual BTW done bit" %
%   B13:0/1  "Service the BTW status / BTW pending" %
%   N14:23/15  "Virtual BTW enable bit" %
%   B13:0/3  "Check BTW Status until done bit is off" %

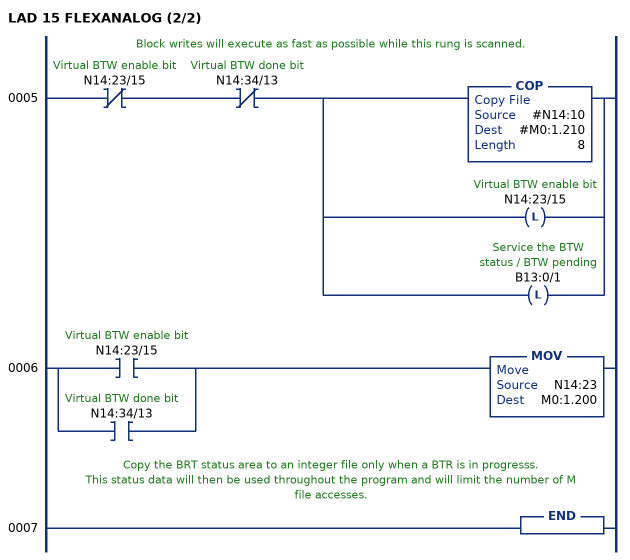
% Rung: 5 %
% Block writes will execute as fast as possible while this rung is scanned. %
SOR XIO N14:23/15 XIO N14:34/13 BST COP #N14:10 #M0:1.210 8 NXB OTL N14:23/15 NXB OTL B13:0/1 BND EOR
%   N14:23/15  "Virtual BTW enable bit" %
%   N14:34/13  "Virtual BTW done bit" %
%   N14:10  "BTW Data" %
%   B13:0/1  "Service the BTW status / BTW pending" %
% Rung: 6 %
SOR BST XIC N14:23/15 NXB XIC N14:34/13 BND MOV N14:23 M0:1.200 EOR
%   N14:23/15  "Virtual BTW enable bit" %
%   N14:34/13  "Virtual BTW done bit" %
% Rung: 7 %
% Copy the BRT status area to an integer file only when a BTR is in progresss.
% This status data will then be used throughout the program and will limit the number of M file accesses. %
SOR END EOR

OTHER DOCUMENTED ADDRESSES
  B3:0/10  LIFT_SPEED_MAN_OVRID  "Used to overide MCP lift speed from the lift controls."
  B3:1/6  MCP_CONT_SLIT_DR
  B3:1/7  PLC_CONT_SLIT_DR
  B3:1/10  MCP_CONT_SLIT_HD
  B3:1/11  PLC_CONT_SLIT_HD
  B3:4/1  PLC_CONT_SLIT_DR_OSR
  B3:4/3  PLC_CONT_SLIT_HD_OSR
  B3:4/8  MCP_CONT_SLIT_DR_OS1
  B3:4/9  MCP_CONT_SLIT_DR_OS2
  B3:4/10  MCP_CONT_SLIT_DR_OS3
  B3:4/11  MCP_CONT_SLIT_DR_OS4
  B3:4/12  PLC_CONT_SLIT_DR_OPN
  B3:4/13  PLC_CONT_SLIT_DR_CLS
  B3:5/0  MCP_CONT_SLIT_HD_OS1
  B3:5/1  MCP_CONT_SLIT_HD_OS2
  B3:5/2  MCP_CONT_SLIT_HD_OS3
  B3:5/3  MCP_CONT_SLIT_HD_OS4
  B3:5/4  PLC_CONT_SLIT_HD_UNL
  B3:5/5  PLC_CONT_SLIT_HD_LTH
  B3:13/15  SPARE_B3_13_15
  B3:14/9  SPARE_B3_14_9
  B3:14/10  SPARE_B3_14_10
  B3:14/11  SPARE_B3_14_11
  B3:14/12  SPARE_B3_14_12
  B3:14/13  SPARE_B3_14_13
  B3:14/14  SPARE_B3_14_14
  B3:14/15  SPARE_B3_14_15
  B3:15/0  SPARE_B3_15_0
  B3:15/1  SPARE_B3_15_1
  B3:15/2  SPARE_B3_15_2
  B3:15/3  SPARE_B3_15_3
  B3:15/4  SPARE_B3_15_4
  B3:15/5  SPARE_B3_15_5
  B3:15/6  SPARE_B3_15_6
  B3:15/7  SPARE_B3_15_7
  B3:15/8  SPARE_B3_15_8
  B3:15/9  SPARE_B3_15_9
  B3:16/0  SPARE_B3_16_0
  B3:16/1  SPARE_B3_16_1
  B3:16/2  SPARE_B3_16_2
  B3:16/3  SPARE_B3_16_3
  B3:16/4  SPARE_B3_16_4
  B3:16/5  SPARE_B3_16_5
  B3:16/6  SPARE_B3_16_6
  B3:16/7  SPARE_B3_16_7
  B3:16/8  SPARE_B3_16_8
  B3:16/9  SPARE_B3_16_9
  B3:16/10  SPARE_B3_16_10
  B3:16/11  SPARE_B3_16_11
  B3:16/12  SPARE_B3_16_12
  B3:16/13  SPARE_B3_16_13
  B3:16/14  SPARE_B3_16_14
  B3:16/15  SPARE_B3_16_15
  B3:17/0  SPARE_B3_17_0
  B3:17/1  SPARE_B3_17_1
  B3:17/2  SPARE_B3_17_2
  B3:17/3  SPARE_B3_17_3
  B3:17/4  SPARE_B3_17_4
  B3:17/5  SPARE_B3_17_5
  B3:17/6  SPARE_B3_17_6
  B3:17/7  SPARE_B3_17_7
  B3:17/8  SPARE_B3_17_8
  B3:17/9  SPARE_B3_17_9
  B3:17/10  SPARE_B3_17_10
  B3:17/11  SPARE_B3_17_11
  B3:17/12  SPARE_B3_17_12
  B3:17/13  SPARE_B3_17_13
  B3:17/14  SPARE_B3_17_14
  B3:17/15  SPARE_B3_17_15
  B3:18/0  SPARE_B3_18_0
  B3:18/1  SPARE_B3_18_1
  B3:18/2  SPARE_B3_18_2
  B3:18/3  SPARE_B3_18_3
  B3:18/4  SPARE_B3_18_4
  B3:18/5  SPARE_B3_18_5
  B3:18/6  SPARE_B3_18_6
  B3:18/7  SPARE_B3_18_7
  B3:18/8  SPARE_B3_18_8
  B3:18/9  SPARE_B3_18_9
  B3:18/10  SPARE_B3_18_10
  B3:18/11  SPARE_B3_18_11
  B3:18/12  SPARE_B3_18_12
  B3:18/13  SPARE_B3_18_13
  B3:18/14  SPARE_B3_18_14
  B3:18/15  SPARE_B3_18_15
  B3:19/0  SPARE_B3_19_0
  B3:19/1  SPARE_B3_19_1
  B3:19/2  SPARE_B3_19_2
  B3:19/3  SPARE_B3_19_3
  B3:19/4  SPARE_B3_19_4
  B3:19/5  SPARE_B3_19_5
  B3:19/6  SPARE_B3_19_6
  B3:19/7  SPARE_B3_19_7
  B3:19/8  SPARE_B3_19_8
  B3:19/9  SPARE_B3_19_9
  B3:19/10  SPARE_B3_19_10
  B3:19/11  SPARE_B3_19_11
  B3:19/12  SPARE_B3_19_12
  B3:19/13  SPARE_B3_19_13
  B3:19/14  SPARE_B3_19_14
  B3:19/15  SPARE_B3_19_15
  B10:0/0  MCP_LIFT_HIGH_PSI  "MCP command to turn on the high lift pressure for camera exchange for the instrument lift."
  B10:0/1  MCP_LIFT_UP_4  "Part of the binary code for up lift speed."
  B10:0/2  MCP_LIFT_UP_3  "Part of the binary code for up lift speed."
  B10:0/3  MCP_LIFT_UP_2  "Part of the binary code for up lift speed."
  B10:0/4  MCP_LIFT_UP_1  "Part of the binary code for up lift speed."
  B10:0/5  MCP_LIFT_DN_1  "Part of the binary code for down lift speed."
  B10:0/6  MCP_LIFT_DN_2  "Part of the binary code for down lift speed."
  B10:0/7  MCP_LIFT_DN_3  "Part of the binary code for down lift speed."
  B10:0/8  MCP_LIFT_DN_4  "Part of the binary code for down lift speed."
  B10:0/9  MCP_PUMP_ON  "MCP command to turn on the instrument lift pump."
  B10:0/10  MCP_SOLENOID_ENGAGE  "MCP command to turn on the instrument lift solenoid.  The solenoid must be on for the lift to work"
  B10:1/1  MCP_15DEG_STOP_EXT_C  "MCP 15 degree stop insert command"
  B10:1/2  MCP_15DEG_STOP_RET_C  "MCP 15 degree stop remove command"
  B10:2/2  MCP_PURGE_CELL_ON  "MCP command to start the purge cell."
  B10:2/3  MCP_PRI_LATCH_CLS_CM  "MCP command to close the primary latches."
  B10:2/4  MCP_PRI_LATCH_OPN_CM  "MCP command to open the primary latches."
  B10:2/5  MCP_SEC_LATCH_CLS_CM  "MCP command to close the secondary latches."
  B10:2/6  MCP_SEC_LATCH_OPN_CM  "MCP command to open the secondary latches."
  B10:2/7  MCP_SAD_LATCH_CLS_CM  "MCP command to close the saddle latches."
  B10:2/8  MCP_SAD_LATCH_OPN_CM  "MCP command to open the saddle latches."
  B10:2/9  MCP_INST_CHG_PROMPT  "MCP command to alert the observers for an instrument change prompt."
  B10:2/10  MCP_INST_CHG_ALERT  "MCP command to alert the observers for an instrument change malfunction."
  B13:0/0  "Servie the BTR status / BTR pending"
  B13:0/2  "Check BTR status until done bit is off"
  DFILE:13  "B13"
  DFILE:14  "N14"
  F8:50  ALT_30D0_LIMIT
  I:1.0/0  INST_LIFT_PUMP_ON  "Instrument lift pump on status bit."
  I:1.0/6  INST_LIFT_MAN  "Instrument lift in the manual mode status bit."
  I:1.0/7  INST_LIFT_HIGH_FORCE  "Instrument lift in high force status bit."
  I:1.0/8  INST_LIFT_LOW_FORCE  "Instrument lift in low force status bit."
  I:1.0/11  OPS_CART_IN_POS  "Imager cart in position status bit."
  I:1.0/12  RACK_0_GRP_0_BIT_12  "Spare input bit"
  I:1.0/15  RACK_0_GRP_0_BIT_15  "Spare PLC input bit."
  I:1.1/0  DOG_HOUSE_CW_PAD  "Dog house cw bump switch.  Stops telescope and windscreen motion if dog house hits obj."
  I:1.1/1  DOG_HOUSE_CCW_PAD  "Dog house ccw bump switch.  Stops telescope and windscreen motion if dog house hits obj."
  I:1.1/2  DOG_HOUSE_DOOR_OPN  "Dog house door open status bit."
  I:1.1/3  DOG_HOUSE_DOOR_CLS  "Dog house door closed status bit."
  I:1.1/4  OPS_CART_IN_HOUSE  "Imager operations cart in dog house status bit."
  I:1.1/5  OPTICAL_BENCH_OPN  "T Bar latches open or off t bars. CCD's safe to move camera."
  I:1.1/6  OPTICAL_BENCH_CLS  "T Bar latches closed or on t bars. CCD's unsafe to move camera."
  I:1.1/7  RACK_0_GRP_1_BIT_7  "Spare PLC input bit."
  I:1.1/8  RACK_0_GRP_1_BIT_8  "Spare PLC input bit."
  I:1.1/9  RACK_0_GRP_1_BIT_9  "Spare PLC input bit."
  I:1.1/15  LOW_LVL_LIGHT_REQ  "Low lever lighting request to change state of low level lighting from off to on or on to off."
  I:1.2/15  SPARE_I1_L1  "MCP Place Holder. Not used in logic code."
  I:1.4/15  SPARE_I1_L2  "MCP Place Holder. Not used in logic code."
  I:1.6/15  SPARE_I1_L3  "MCP Place Holder. Not used in logic code."
  I:1.8/14  CLOSE_SLIT_DOORS  "Latch control box Slithead door Close switch"
  I:1.8/15  OPEN_SLIT_DOORS  "Latch control box Slithead door Open switch"
  I:1.9/0  SLIT_LATCH_UNLTH_CMD  "Slit head unlatch command input"
  I:1.9/1  SLIT_LATCH_LTH_CMD  "Slit head latch command input"
  I:1.9/4  RACK_1_GRP_1_BIT_4  "Spare PLC input bit."
  I:1.9/5  RACK_1_GRP_1_BIT_5  "Spare PLC input bit."
  I:1.9/6  RACK_1_GRP_1_BIT_6  "Spare PLC input bit."
  I:1.9/7  RACK_1_GRP_1_BIT_7  "Spare PLC input bit."
  I:1.9/8  RACK_1_GRP_1_BIT_8  "Spare PLC input bit."
  I:1.9/9  RACK_1_GRP_1_BIT_9  "Spare PLC input bit."
  I:1.9/10  RACK_1_GRP_1_BIT_10  "Spare PLC input bit."
  I:1.9/11  RACK_1_GRP_1_BIT_11  "Spare PLC input bit."
  I:1.9/12  RACK_1_GRP_1_BIT_12  "Spare PLC input bit."
  I:1.9/13  RACK_1_GRP_1_BIT_13  "Spare PLC input bit."
  I:1.9/14  RACK_1_GRP_1_BIT_14  "Spare PLC input bit."
  I:1.9/15  RACK_1_GRP_1_BIT_15  "Spare PLC input bit."
  I:1.10/15  SPARE_I1_L5  "MCP Place Holder. Not used in logic code."
  I:1.12/15  SPARE_I1_L6  "MCP Place Holder. Not used in logic code."
  I:1.14/15  SPARE_I1_L7  "MCP Place Holder. Not used in logic code."
  I:1.16/15  RACK_2_GRP_0_BIT_15  "Spare PLC input bit."
  I:1.18/0  SAD_LATCH1_OPN  "Saddle latch 1 open status."
  I:1.18/2  SAD_LATCH2_OPN  "Saddle latch 2 open status."
  I:1.18/14  RACK_2_GRP_2_BIT_14  "Spare PLC input bit."
  I:1.18/15  RACK_2_GRP_2_BIT_15  "Spare PLC input bit."
  I:1.20/0  PURGE_AIR_PRESSUR_SW  "Purge air pressure switch"
  I:1.20/3  SEC_MIR_FORCE_LIMITS  "Secondary Mirror Force Limit bit."
  I:1.20/4  RACK_2_GRP_4_BIT_4  "Spare PLC input bit."
  I:1.20/5  RACK_2_GRP_4_BIT_5  "Spare PLC input bit."
  I:1.20/6  RACK_2_GRP_4_BIT_6  "Spare PLC input bit."
  I:1.20/7  RACK_2_GRP_4_BIT_7  "Spare PLC input bit."
  I:1.20/8  RACK_2_GRP_4_BIT_8  "Spare PLC input bit."
  I:1.20/9  RACK_2_GRP_4_BIT_9  "Spare PLC input bit."
  I:1.20/10  RACK_2_GRP_4_BIT_10  "Spare PLC input bit."
  I:1.20/11  RACK_2_GRP_4_BIT_11  "Spare PLC input bit."
  I:1.20/12  RACK_2_GRP_4_BIT_12  "Spare PLC input bit."
  I:1.20/13  RACK_2_GRP_4_BIT_13  "Spare PLC input bit."
  I:1.20/14  RACK_2_GRP_4_BIT_14  "Spare PLC input bit."
  I:1.20/15  RACK_2_GRP_4_BIT_15  "Spare PLC input bit."
  I:1.22/15  SPARE_I1_L11  "MCP Place Holder. Not used in logic code."
  I:1.24/15  SPARE_I1_L12  "MCP Place Holder. Not used in logic code."
  I:1.25/0  RACK_3_GRP_1_BIT_0  "Spare PLC input bit."
  I:1.25/10  RACK_3_GRP_1_BIT_10  "Spare PLC input bit."
  I:1.25/11  RACK_3_GRP_1_BIT_11  "Spare PLC input bit."
  I:1.25/12  RACK_3_GRP_1_BIT_12  "Spare PLC input bit."
  I:1.25/13  RACK_3_GRP_1_BIT_13  "Spare PLC input bit."
  I:1.25/14  RACK_3_GRP_1_BIT_14  "Spare PLC input bit."
  I:1.25/15  RACK_3_GRP_1_BIT_15  "Spare PLC input bit."
  I:1.26  SCREEN_STATUS  "FF Screen status word"
  I:1.26/0  LEAF_1_OPEN_STAT  "Leaf Screen 1 open status bit"
  I:1.26/2  LEAF_2_OPEN_STAT  "Leaf Screen 2 open status bit"
  I:1.26/4  LEAF_3_OPEN_STAT  "Leaf Screen 3 open status bit"
  I:1.26/6  LEAF_4_OPEN_STAT  "Leaf Screen 4 open status bit"
  I:1.26/8  LEAF_5_OPEN_STAT  "Leaf Screen 5 open status bit"
  I:1.26/10  LEAF_6_OPEN_STAT  "Leaf Screen 6 open status bit"
  I:1.26/12  LEAF_7_OPEN_STAT  "Leaf Screen 7 open status bit"
  I:1.26/14  LEAF_8_OPEN_STAT  "Leaf Screen 8 open status bit"
  I:1.27  LAMP_STATUS  "Flatfield Lamp Status Word"
  I:1.27/0  FF_1_STAT  "Flatfield lamp 1 status bit"
  I:1.27/1  FF_2_STAT  "Flatfield lamp 2 status bit"
  I:1.27/2  FF_3_STAT  "Flatfield lamp 3 status bit"
  I:1.27/3  FF_4_STAT  "Flatfield lamp 4 status bit"
  I:1.27/4  NE_1_STAT  "Neon lamp 1 status bit"
  I:1.27/5  NE_2_STAT  "Neon lamp 2 status bit"
  I:1.27/6  NE_3_STAT  "Neon lamp 3 status bit"
  I:1.27/7  NE_4_STAT  "Neon lamp 4 status bit"
  I:1.27/8  HGCD_1_STAT  "Mercury-cadmium lamp 1 status bit"
  I:1.27/9  HGCD_2_STAT  "Mercury-cadmium lamp 2 status bit"
  I:1.27/10  HGCD_3_STAT  "Mercury-cadmium lamp 3 status bit"
  I:1.27/11  HGCD_4_STAT  "Mercury-cadmium lamp 4 status bit"
  I:1.27/12  RACK_3_GRP_3_BIT_12  "Spare PLC input bit."
  I:1.27/13  RACK_3_GRP_3_BIT_13  "Spare PLC input bit."
  I:1.27/14  RACK_3_GRP_3_BIT_14  "Spare PLC input bit."
  I:1.27/15  RACK_3_GRP_3_BIT_15  "Spare PLC input bit."
  I:1.28/8  RACK_3_GRP_4_BIT_8  "Spare PLC input bit."
  I:1.28/9  RACK_3_GRP_4_BIT_9  "Spare PLC input bit."
  I:1.28/10  RACK_3_GRP_4_BIT_10  "Spare PLC input bit."
  I:1.28/11  RACK_3_GRP_4_BIT_11  "Spare PLC input bit."
  I:1.28/12  RACK_3_GRP_4_BIT_12  "Spare PLC input bit."
  I:1.28/13  RACK_3_GRP_4_BIT_13  "Spare PLC input bit."
  I:1.28/14  RACK_3_GRP_4_BIT_14  "Spare PLC input bit."
  I:1.28/15  RACK_3_GRP_4_BIT_15  "Spare PLC input bit."
  I:1.30/15  SPARE_I1_L15  "MCP Place Holder. Not used in logic code."
  I:2.1  WIND_DC_INPUT_CARD  "Windscreen digital input card values."
  I:2.1/0  WIND_AZ1_FAULT  "Windscreen azimuth amplifier 1 fault bit."
  I:2.1/1  WIND_AZ2_FAULT  "Windscreen azimuth amplifier 2 fault bit."
  I:2.1/2  WIND_AZ3_FAULT  "Windscreen azimuth amplifier 3 fault bit."
  I:2.1/3  WIND_ALT1_FAULT  "Windscreen altitude amplifier fault bit."
  I:2.1/4  WIND_AZ_PERM  "Windscreen azimuth motion permit bit."
  I:2.1/5  WIND_ALT_PERM  "Windscreen altitude motion permit bit."
  I:2.1/15  SPARE  "Spare PLC input bit."
  I:2.2  AZ_PID_STATUS  "Azimuth PID Status Word"
  I:2.3  AZ_LVDT_ERROR  "Azimuth LVDT error analog value."
  I:2.4  AZ_PRI_DRV  "Azimuth primary drive value."
  I:2.5  AZ_FEED_FWD_DRV  "Azimuth feed forward drive value."
  I:2.6  DCM_1_WORD6_SPARE  "DCM 1 spare word"
  I:2.7  DCM_1_WORD7_SPARE  "DCM 1 spare word"
  I:2.8  DCM_2_STATUS_WORD  "Direct communications module 2 status word."
  I:2.9  DCM_2_WORD1_SPARE  "DCM 2 spare word"
  I:2.10  ALT_PID_STATUS  "Altitude PID Status Word"
  I:2.11  ALT_LVDT_ERROR  "Altitude LVDT error analog value."
  I:2.12  ALT_PRI_DRV  "Altitude primary drive value."
  I:2.13  DCM_2_WORD5_SPARE  "DCM 2 spare word"
  I:2.14  DCM_2_WORD6_SPARE  "DCM 2 spare word"
  I:2.15  DCM_2_WORD7_SPARE  "DCM 2 spare word"
  I:3.1  AZ_1_CURRENT  "Azimuth motor 1 current."
  I:3.2  AZ_2_VOLTAGE  "Azimuth motor 2 voltage."
  I:3.3  AZ_2_CURRENT  "Azimuth motor 2 current."
  I:3.5  ALT_1_CURRENT  "Altitude motor 1 current."
  I:3.6  ALT_2_VOLTAGE  "Altitude motor 2 voltage."
  I:3.7  ALT_2_CURRENT  "Altitude motor 2 current."
  I:4.2  ROT_1_CURRENT  "Rotator motor current."
  I:4.3  UMBILICAL_DIST  "Camera umbilical distance value."
  I:4.6  I_4_ANALOG_6_SPARE  "Spare analog channel."
  I:4.7  I_4_ANALOG_7_SPARE  "Spare analog channel."
  I:5.1  COUNTERWEIGHT_2_POS  "Counterweight #2 string pot position value"
  I:5.2  COUNTERWEIGHT_3_POS  "Counterweight #3 string pot position value"
  I:5.3  COUNTERWEIGHT_4_POS  "Counterweight #4 string pot position value"
  I:5.4  I_5_ANALOG_4_SPARE  "Spare analog channel."
  I:5.5  I_5_ANALOG_5_SPARE  "Spare analog channel."
  I:5.6  I_5_ANALOG_6_SPARE  "Spare analog channel."
  I:5.7  I_5_ANALOG_7_SPARE  "Spare analog channel."
  I:6.0/0  TCC_STOP  "TCC inhibit input hook.  Currently not implemented."
  I:6.0/2  SPARE_S1_C2  "Spare splitter chassis channel."
  I:6.0/3  FIBER_SIGNAL_LOSS  "Control room e-stop fiber link signal loss indicator. Currently not implemented."
  I:6.0/15  MCP_WATCHDOG_TIMER  "MCP Watchdog Timer. Removes drive amplifier reference if MCP Fault."
  I:6.1/2  ALT_MTR1_PERM_IN  "Altitude motor 1 permit status"
  I:6.1/3  ALT_MTR2_PERM_IN  "Altitude motor 2 permit status"
  I:6.1/4  WIND_ALT_MTR_PERM_IN  "Wind screen altitude motor permit in"
  I:6.1/5  ALT_PLC_PERM_IN  "Altitude PLC permit status"
  I:6.1/6  WIND_ALT_PLC_PERM_IN  "Wind screen PLC permit status"
  I:6.1/7  AZ_STOW_3A  "Azimuth stow position switch status"
  I:6.1/10  AZ_MTR1_PERM_IN  "Azimuth motor 1 permit status"
  I:6.1/11  AZ_MTR2_PERM_IN  "Azimuth motor 2 permit status"
  I:6.1/12  WIND_AZ_MTR_PERM_IN  "Wind screen azimuth motor permit status"
  I:6.1/13  AZ_PLC_PERM_IN  "Azimuth PLC permit status"
  I:6.1/14  WIND_AZ_PLC_PERM_IN  "Wind screen PLC permit status"
  I:6.1/15  AZ_STOW_3B  "Azimuth stow position switch status"
  I:7.0/0  ROT_MTR_CW_PERM_IN  "Rotator motor CW permit status"
  I:7.0/1  ROT_MTR_CCW_PERM_IN  "Rotator motor CCW permit status"
  I:7.0/2  ROT_MTR_PERM_IN  "Rotator motor permit status"
  I:7.0/3  SPARE_S5_C3  "Spare splitter chassis channel"
  I:7.0/4  BLDG_PERM_IN  "Building motion permit status"
  I:7.0/5  ROT_PLC_PERM_IN  "Rotator PLC permit status"
  I:7.0/6  HATCH_CLS  "Hatch closed status switch"
  I:7.0/8  ALT_GRT_0D3_LIMIT  "Altitude greater then 0.3 degree limit status"
  I:7.0/10  ALT_LES_90D5_LIMIT  "Altitude less than 90.5 degree limit status"
  I:7.0/12  AZ_109_131_LIMIT_1  "Azimuth between 109 to 131 degrees status"
  I:7.0/13  ALT_GRT_18D6_LIMIT_1  "Altitude greater than 18.6 degree limit status"
  I:7.1/0  ALT_GRT_83_LIMIT_1  "Altitude greater than 83 degree limit status"
  I:7.1/5  ALT_GRT_18D6_LIMIT_2  "Altitude greater than 18.6 degree limit status"
  I:7.1/6  ALT_SLIP  "Altitude slip detection status"
  I:7.1/7  ALT_VELOCITY_LIMIT  "Altitude velocity limit status"
  I:7.1/10  AZ_NEG_201A_CW  "Azimuth greater then -201 degrees status"
  I:7.1/11  AZ_POS_445A_CCW  "Azimuth less than +445 degree limit status"
  I:7.1/12  AZ_NEG_201B_CW  "Azimuth greater than -201 degrees status"
  I:7.1/13  AZ_POS_445B_CCW  "Azimuth less than +445 degree limit status"
  I:7.1/14  SPARE_S8_C6  "Spare splitter chassis channel"
  I:7.1/15  SPARE_S8_C7  "Spare splitter chassis channel"
  I:8.0/0  ALT_GRT_18D6_LIMIT_3  "Altitude greater than 18.6 degree limit status"
  I:8.0/1  BLDG_ON_AZ  "Building on status for Azimuth logic"
  I:8.0/2  AZ_109_131_LIMIT_2  "Azimuth between 109 and 131 degrees limit status"
  I:8.0/3  ALT_GRT_83_LIMIT_2  "Altitude greater then 83 degree limit status"
  I:8.0/5  SPARE_S9_C5  "Spare splitter chassis channel"
  I:8.0/6  AZ_SLIP  "Azimuth slip detection status"
  I:8.0/7  AZ_VELOCITY_LIMIT  "Azimuth velocity limit status"
  I:8.0/10  ROT_NEG_200A_CW  "Rotator greater then -200 degrees status"
  I:8.0/11  ROT_POS_380A_CCW  "Rotator less than +300 degree limit status"
  I:8.0/12  ROT_NEG_200B_CW  "Rotator greater then -200 degrees status"
  I:8.0/13  ROT_POS_380B_CCW  "Rotator less than +300 degree limit status"
  I:8.0/14  ROT_SLIP  "Rotator slip detection status"
  I:8.0/15  ROT_VELOCITY_LIMIT  "Rotator velocity limit status"
  I:8.1/9  UMBILICAL_STRAIN_SW  "Camera umbilical strain switch status"
  I:8.1/12  IN_8_BIT_28_SPARE  "Spare PLC Input Bit"
  I:8.1/13  IN_8_BIT_29_SPARE  "Spare PLC Input Bit"
  I:9.0/3  AZ_BRAKE_EN_STAT  "Azimuth brake enabled status"
  I:9.0/10  IN_9_BIT_10_SPARE  "Spare PLC Input Bit"
  I:9.0/11  IN_9_BIT_11_SPARE  "Spare PLC Input Bit"
  I:9.0/12  IN_9_BIT_12_SPARE  "Spare PLC Input Bit"
  I:9.0/13  IN_9_BIT_13_SPARE  "Spare PLC Input Bit"
  I:9.0/14  IN_9_BIT_14_SPARE  "Spare PLC Input Bit"
  I:9.0/15  IN_9_BIT_15_SPARE  "Spare PLC Input Bit"
  I:9.1/0  S1_C0_BYPASS_SW  "E-Stop bypass monitor status"
  I:9.1/1  S1_C1_BYPASS_SW  "E-Stop bypass monitor status"
  I:9.1/2  S1_C2_BYPASS_SW  "E-Stop bypass monitor status"
  I:9.1/3  S1_C3_BYPASS_SW  "E-Stop bypass monitor status"
  I:9.1/15  S2_C7_MCP_WTCHDG_BYP  "MCP watchdog bypass monitor status"
  I:10.0/0  IN_10_BIT_0_SPARE  "Spare PLC Input Bit"
  I:10.0/1  IN_10_BIT_1_SPARE  "Spare PLC Input Bit"
  I:10.0/2  IN_10_BIT_2_SPARE  "Spare PLC Input Bit"
  I:10.0/3  IN_10_BIT_3_SPARE  "Spare PLC Input Bit"
  I:10.0/4  IN_10_BIT_4_SPARE  "Spare PLC Input Bit"
  I:10.0/5  IN_10_BIT_5_SPARE  "Spare PLC Input Bit"
  I:10.0/6  IN_10_BIT_6_SPARE  "Spare PLC Input Bit"
  I:10.0/7  IN_10_BIT_7_SPARE  "Spare PLC Input Bit"
  I:10.0/8  IN_10_BIT_8_SPARE  "Spare PLC Input Bit"
  I:10.0/9  IN_10_BIT_9_SPARE  "Spare PLC Input Bit"
  I:10.0/10  IN_10_BIT_10_SPARE  "Spare PLC Input Bit"
  I:10.0/11  IN_10_BIT_11_SPARE  "Spare PLC Input Bit"
  I:10.0/12  IN_10_BIT_12_SPARE  "Spare PLC Input Bit"
  I:10.0/13  IN_10_BIT_13_SPARE  "Spare PLC Input Bit"
  I:10.0/14  IN_10_BIT_14_SPARE  "Spare PLC Input Bit"
  I:10.0/15  IN_10_BIT_15_SPARE  "Spare PLC Input Bit"
  I:10.1/0  IN_10_BIT_16_SPARE  "Spare PLC Input Bit"
  I:10.1/1  IN_10_BIT_17_SPARE  "Spare PLC Input Bit"
  I:10.1/2  IN_10_BIT_18_SPARE  "Spare PLC Input Bit"
  I:10.1/3  IN_10_BIT_19_SPARE  "Spare PLC Input Bit"
  I:10.1/4  IN_10_BIT_20_SPARE  "Spare PLC Input Bit"
  I:10.1/5  IN_10_BIT_21_SPARE  "Spare PLC Input Bit"
  I:10.1/6  IN_10_BIT_22_SPARE  "Spare PLC Input Bit"
  I:10.1/7  IN_10_BIT_23_SPARE  "Spare PLC Input Bit"
  I:10.1/8  IN_10_BIT_24_SPARE  "Spare PLC Input Bit"
  I:10.1/9  IN_10_BIT_25_SPARE  "Spare PLC Input Bit"
  I:10.1/10  IN_10_BIT_26_SPARE  "Spare PLC Input Bit"
  I:10.1/11  IN_10_BIT_27_SPARE  "Spare PLC Input Bit"
  I:10.1/12  IN_10_BIT_28_SPARE  "Spare PLC Input Bit"
  I:10.1/13  IN_10_BIT_29_SPARE  "Spare PLC Input Bit"
  I:10.1/14  IN_10_BIT_30_SPARE  "Spare PLC Input Bit"
  I:10.1/15  IN_10_BIT_31_SPARE  "Spare PLC Input Bit"
  M00000:001.100  "BTR control bits"
  M00000:001.200  "BTW Control"
  M00000:001.210  "BTW Data"
  N14:0  "BTR Data"
  N14:20/15  "Virtual BTR Enable bit"
  N14:30  "BTR Status"
  N14:30/13  "Virtual BTR Done Bit"
  O:1.0/15  SPARE_O1_L0  "MCP Place Holder. Not used in logic code."
  O:1.2/0  INST_LIFT_HIGH_PSI  "Instrument lift high pressure enable bit"
  O:1.4/15  SPARE_O1_L2  "MCP Place Holder. Not used in logic code."
  O:1.6/15  SPARE_01_L3  "MCP Place Holder. Not used in logic code."
  O:1.8/15  SPARE_O1_L4  "MCP Place Holder. Not used in logic code."
  O:1.10/10  DOG_DOOR_OPEN_LED  "Dog house door not closed LED"
  O:1.10/11  CAM_CRT_IN_HOUSE_LED  "Camera cart in dog house LED"
  O:1.13/13  RACK_1_GRP_5_BIT_13  "Spare PLC output bit."
  O:1.13/14  RACK_1_GRP_5_BIT_14  "Spare PLC output bit."
  O:1.13/15  RACK_1_GRP_5_BIT_15  "Spare PLC output bit."
  O:1.14/15  SPARE_O1_L7  "MCP Place Holder. Not used in logic code."
  O:1.16/15  SPARE_O1_L8  "MCP Place Holder. Not used in logic code."
  O:1.18/15  SPARE_O1_L9  "MCP Place Holder. Not used in logic code."
  O:1.19/6  RACK_2_GRP_3_BIT_6  "Spare PLC output bit."
  O:1.19/7  RACK_2_GRP_3_BIT_7  "Spare PLC output bit."
  O:1.19/8  RACK_2_GRP_3_BIT_8  "Spare PLC output bit."
  O:1.19/9  RACK_2_GRP_3_BIT_9  "Spare PLC output bit."
  O:1.19/10  RACK_2_GRP_3_BIT_10  "Spare PLC output bit."
  O:1.19/11  RACK_2_GRP_3_BIT_11  "Spare PLC output bit."
  O:1.19/12  RACK_2_GRP_3_BIT_12  "Spare PLC output bit."
  O:1.19/13  RACK_2_GRP_3_BIT_13  "Spare PLC output bit."
  O:1.19/14  RACK_2_GRP_3_BIT_14  "Spare PLC output bit."
  O:1.19/15  RACK_2_GRP_3_BIT_15  "Spare PLC output bit."
  O:1.20/15  SPARE_O1_L10  "MCP Place Holder. Not used in logic code."
  O:1.21/1  RACK_2_GRP_5_BIT_1  "Spare PLC output bit."
  O:1.21/2  RACK_2_GRP_5_BIT_2  "Spare PLC output bit."
  O:1.21/3  RACK_2_GRP_5_BIT_3  "Spare PLC output bit."
  O:1.21/4  RACK_2_GRP_5_BIT_4  "Spare PLC output bit."
  O:1.21/5  RACK_2_GRP_5_BIT_5  "Spare PLC output bit."
  O:1.21/6  RACK_2_GRP_5_BIT_6  "Spare PLC output bit."
  O:1.21/7  RACK_2_GRP_5_BIT_7  "Spare PLC output bit."
  O:1.21/8  RACK_2_GRP_5_BIT_8  "Spare PLC output bit."
  O:1.21/9  RACK_2_GRP_5_BIT_9  "Spare PLC output bit."
  O:1.21/10  RACK_2_GRP_5_BIT_10  "Spare PLC output bit."
  O:1.21/11  RACK_2_GRP_5_BIT_11  "Spare PLC output bit."
  O:1.21/12  RACK_2_GRP_5_BIT_12  "Spare PLC output bit."
  O:1.21/13  RACK_2_GRP_5_BIT_13  "Spare PLC output bit."
  O:1.21/14  RACK_2_GRP_5_BIT_14  "Spare PLC output bit."
  O:1.21/15  AUDIO_WARNING_2  "Audio warning used for instrument change error"
  O:1.22/15  SPARE_O1_L11  "MCP Place Holder. Not used in logic code."
  O:1.24/15  SPARE_O1_L12  "MCP Place Holder. Not used in logic code."
  O:1.26/15  SPARE_O1_L13  "MCP Place Holder. Not used in logic code."
  O:1.28/15  SPARE_O1_L14  "MCP Place Holder. Not used in logic code."
  O:1.29  FLAT_FIELD_CONTROL  "Flatfield screen control word"
  O:1.29/9  RACK_4_GRP_5_BIT_9  "Spare PLC output bit."
  O:1.29/10  RACK_4_GRP_5_BIT_10  "Spare PLC output bit."
  O:1.29/11  RACK_4_GRP_5_BIT_11  "Spare PLC output bit."
  O:1.29/12  RACK_4_GRP_5_BIT_12  "Spare PLC output bit."
  O:1.29/13  RACK_4_GRP_5_BIT_13  "Spare PLC output bit."
  O:1.29/14  RACK_4_GRP_5_BIT_14  "Spare PLC output bit."
  O:1.29/15  AUDIO_WARNING_1  "Audio warning used for instrument change error"
  O:1.30/15  SPARE_O1_L15  "MCP Place Holder. Not used in logic code."
  O:2.1/4  OUT_2_BIT_20_SPARE  "Spare PLC output bit."
  O:2.1/5  OUT_2_BIT_21_SPARE  "Spare PLC output bit"
  O:11.1/8  OUT_11_BIT_24_SPARE  "Spare PLC output bit."
  O:11.1/9  OUT_11_BIT_25_SPARE  "Spare PLC output bit."
  O:11.1/11  OUT_11_BIT_27_SPARE  "Spare PLC output bit."
  O:12.0/13  OUT_12_BIT_13_SPARE  "Spare PLC Output Bit"
  O:12.0/14  OUT_12_BIT_14_SPARE  "Spare PLC Output Bit"
  O:12.0/15  OUT_12_BIT_15_SPARE  "Spare PLC Output Bit"
  O:12.1/0  OUT_12_BIT_16_SPARE  "Spare PLC Output Bit"
  O:12.1/1  OUT_12_BIT_17_SPARE  "Spare PLC Output Bit"
  O:12.1/2  OUT_12_BIT_18_SPARE  "Spare PLC Output Bit"
  O:12.1/3  OUT_12_BIT_19_SPARE  "Spare PLC Output Bit"
  O:12.1/4  OUT_12_BIT_20_SPARE  "Spare PLC Output Bit"
  O:12.1/5  OUT_12_BIT_21_SPARE  "Spare PLC Output Bit"
  O:12.1/6  OUT_12_BIT_22_SPARE  "Spare PLC Output Bit"
  O:12.1/7  OUT_12_BIT_23_SPARE  "Spare PLC Output Bit"
  O:12.1/8  OUT_12_BIT_24_SPARE  "Spare PLC Output Bit"
  O:12.1/9  OUT_12_BIT_25_SPARE  "Spare PLC Output Bit"
  O:12.1/10  OUT_12_BIT_26_SPARE  "Spare PLC Output Bit"
  O:12.1/11  OUT_12_BIT_27_SPARE  "Spare PLC Output Bit"
  O:12.1/12  OUT_12_BIT_28_SPARE  "Spare PLC Output Bit"
  O:12.1/13  OUT_12_BIT_29_SPARE  "Spare PLC Output Bit"
  O:12.1/14  OUT_12_BIT_30_SPARE  "Spare PLC Output Bit"
  O:12.1/15  OUT_12_BIT_31_SPARE  "Spare PLC Output Bit"
  U:4  "Windscreen Azimuth Axis Motion Control Logic"
  U:6  "Windscreen Altitude Axis Motion Control Logic"

COMMENTS NOT ATTACHED TO A CURRENT RUNG
  RUNG000004-000000: Windscreen Azimuth Axis Motion Control Logic / The following code is used to control the PLC Windscreen Azimuth Axis Permit.
  RUNG000006-000000: Windscreen Altitude Axis Motion Control Logic / The following code is used to control the PLC Telescope Windscreen altitude Axis Permit.
  RUNG000015-000013: Unlatch the bit that continues to check the BTR status.  When a BTR is complete, the done bit is set.  The ladder program must then unlatch the enable bit, then wait for the SN module to turn off the done bit before another BTR to the same M-File location can be initiated.  This is one complete BTR cycle.
  RUNG000015-000014: Copy the BTW status area to an integer file only when a BTW is in progress.
    This status data will then be used throughout the program and will limit the number of M file accesses.
  RUNG000015-000015: Unlatch the bit that continues to check the BTW status.  When a BTW is
    complete, the done bit is set.  The ladder program must then unlatch the enable
    bit, then wait for the SN module to turn off the done bit before another
    BTW to the same M file location can be initiated.  This completes one BTW cycle.
  RUNG000015-000016: When a BTR successfully completes, buffer the BTR data and unlatch the BTR enable bit.  Also, unlatch the BTR pending bit and latch the bit that continues checking the BTR status until the SN module turns off the done bit.
  RUNG000015-000017: When a BTW successfully completes, unlatch the BTW enable bit and the BTW
    pending bit to complete a BTW sequence.  Also, unlatch the bit that continues
    checking the BTW status until the SN module turns the done bit off.
  RUNG000015-000018: Block transfer reads will execute continiously as long as these rungs are scanned.
  RUNG000015-000019: Block writes will execute as fast as possible while this rung is scanned.
  RUNG000015-000020: Move the virtual control word to the M0 file for the SN module whenever a transition of the BTR enable bit occurs.
  RUNG000015-000021: Move the virtual control word to the M0 file for the SN module whenever a transition of the BTR enable bit occurs.
  RUNG000015-000022: Temperature monitoring / The following code is used to aquire the temperature data from the Altitude junction box #2 rtd module 1.
    
    Configure the BTR and BTW operation type, length and RIO address at power up.
    Bit N14:100/7 must be set to indicate a BTR operation and N14:103/7 must be reset to indicate BTW operation.
    
    N14:100 = 128 Set the BTR Read bit, no time out.
    N14:101 = 11 Set the transfer length to 9 words of data
    N14:102 = 160 Set to rack 1 group 6 slot 0
    
    N14:103 = 0 Set the BTW write  bit, no time out.
    N14:104 = 3 Set the transfer length to 3 word of data
    N14:105 = 160 Set to rack 1 group 6 slot 0
  RUNG000015-000023: Copy the BRT status area to an integer file only when a BTR is in progresss.
    This status data will then be used throughout the program and will limit the number of M file accesses.
  RUNG000015-000024: Unlatch the bit that continues to check the BTR status.  When a BTR is complete, the done bit is set.  The ladder program must then unlatch the enable bit, then wait for the SN module to turn off the done bit before another BTR to the same M-File location can be initiated.  This is one complete BTR cycle.
  RUNG000015-000025: Copy the BTW status area to an integer file only when a BTW is in progress.
    This status data will then be used throughout the program and will limit the number of M file accesses.
  RUNG000015-000026: Unlatch the bit that continues to check the BTW status.  When a BTW is
    complete, the done bit is set.  The ladder program must then unlatch the enable
    bit, then wait for the SN module to turn off the done bit before another
    BTW to the same M file location can be initiated.  This completes one BTW cycle.
  RUNG000015-000027: When a BTR successfully completes, buffer the BTR data and unlatch the BTR enable bit.  Also, unlatch the BTR pending bit and latch the bit that continues checking the BTR status until the SN module turns off the done bit.
  RUNG000015-000028: When a BTW successfully completes, unlatch the BTW enable bit and the BTW
    pending bit to complete a BTW sequence.  Also, unlatch the bit that continues
    checking the BTW status until the SN module turns the done bit off.
  RUNG000015-000029: Block transfer reads will execute continiously as long as these rungs are scanned.
  RUNG000015-000030: Block writes will execute as fast as possible while this rung is scanned.
  RUNG000015-000031: Move the virtual control word to the M0 file for the SN module whenever a transition of the BTR enable bit occurs.
  RUNG000015-000032: Move the virtual control word to the M0 file for the SN module whenever a transition of the BTR enable bit occurs.
  RUNG000015-000033: Temperature monitoring / The following code is used to aquire the temperature data from the Altitude junction box #2 rtd module 2.
    
    Configure the BTR and BTW operation type, length and RIO address at power up.
    Bit N14:140/7 must be set to indicate a BTR operation and N14:143/7 must be reset to indicate BTW operation.
    
    N14:140 = 128 Set the BTR Read bit, no time out.
    N14:141 = 11 Set the transfer length to 9 words of data
    N14:142 = 301 Set to rack 1 group 7 slot 0
    
    N14:143 = 0 Set the BTW write  bit, no time out.
    N14:144 = 3 Set the transfer length to 3 word of data
    N14:145 = 301 Set to rack 1 group 7 slot 0
  RUNG000015-000034: Copy the BRT status area to an integer file only when a BTR is in progresss.
    This status data will then be used throughout the program and will limit the number of M file accesses.
  RUNG000015-000035: Unlatch the bit that continues to check the BTR status.  When a BTR is complete, the done bit is set.  The ladder program must then unlatch the enable bit, then wait for the SN module to turn off the done bit before another BTR to the same M-File location can be initiated.  This is one complete BTR cycle.
  RUNG000015-000036: Copy the BTW status area to an integer file only when a BTW is in progress.
    This status data will then be used throughout the program and will limit the number of M file accesses.
  RUNG000015-000037: Unlatch the bit that continues to check the BTW status.  When a BTW is
    complete, the done bit is set.  The ladder program must then unlatch the enable
    bit, then wait for the SN module to turn off the done bit before another
    BTW to the same M file location can be initiated.  This completes one BTW cycle.
  RUNG000015-000038: When a BTR successfully completes, buffer the BTR data and unlatch the BTR enable bit.  Also, unlatch the BTR pending bit and latch the bit that continues checking the BTR status until the SN module turns off the done bit.
  RUNG000015-000039: When a BTW successfully completes, unlatch the BTW enable bit and the BTW
    pending bit to complete a BTW sequence.  Also, unlatch the bit that continues
    checking the BTW status until the SN module turns the done bit off.
  RUNG000015-000040: Block transfer reads will execute continiously as long as these rungs are scanned.
  RUNG000015-000041: Block writes will execute as fast as possible while this rung is scanned.
  RUNG000015-000042: Move the virtual control word to the M0 file for the SN module whenever a transition of the BTR enable bit occurs.
  RUNG000015-000043: Move the virtual control word to the M0 file for the SN module whenever a transition of the BTR enable bit occurs.

REVISION NOTES
  137: added brake and umbilical bits
  138: BRAKE COMMAND AND STATUS ADDED
  139: brake added to azimuth permit ladder
  140: azimuth brake interlock in az motor permit rung
  141: added altitude brake inhibit for altitude motors
  142: added altitude brake inhibit for altitude motors
  146: added doghouse interlock to telescope altitude permit
  272: Modified Alt Position information to degrees vs counts.
     This should make reading the logic code easier.
  359: I/O Modifications
  360: I/O Modifications
  361: Added MCP placeholder bits to the address database.
  364: Updated Version from CVS
  365: Put in new name for I:9/31 (S2_C7_MCP_WTCHDG_BYP - MCP watchdog bypass monitor status)
  366: V23 changes the voltage and current minimums for motor resistance calculations from
     100 to 500 counts (.6 to 3 V), (.2 to 1 A)
  367: Inst ID change
  368: Inst ID change
  369: Changing instrument ID scheme to accommodate BOSS
  370: Instrument ID scheme changed to accommodate BOSS
  371: Change in instrument ID scheme to accommodate new BOSS cartridges
  372: Change in instrument ID scheme to accommodate BOSS
  373: Removing Imager Interlocks now that imager is gone
  374: Imager Interlocks Removal
  375: engcam and corrector now valid combination
  376: Added Cartridge 18
  377: Added Cartridge 18
  378: cartridge 18 logic added
  379: cart 18 logic
  380: Lift Latch Height Adjustment
  381: Lift Latch Height Adjust
  382: Lift Latch Height Adjust
  383: Lowered altitude limit to 18 degrees
  384: Lowered altitude limit to 18 degrees
  385: Lower altitude limit to 18 degrees
  386: DIMM FFS avoidance
  387: FFS DIMM avoidance
  388: FFS DIMM avoidance
  389: Adding logic for gang connector status
  390: Added logic for APOGEE and MARVELS gang connector status and Viktor pin control
  391: Logic added for gang connector status/protection
  392: Added logic for gang connector status/protection
  393: Updated APOGEE gang connector status switches.  Removed MARVELS status switch logic
  394: Updated gang connector status bits
  395: updated gang connector status switches
  396: updated gang connector status bits

DATA TABLE (non-zero values as saved)
DATA T4
% .PRE .ACC %
% T4:0 % 800 0
% T4:1 % 800 0
% T4:2 % 50 0
% T4:3 % 800 0
% T4:4 % 800 0
% T4:5 % 3000 0
% T4:6 % 500 0
% T4:7 % 500 0
% T4:8 % 500 0
% T4:10 % 200 0
% T4:11 % 200 0
% T4:12 % 200 0
% T4:13 % 200 0
% T4:14 % 200 0
% T4:15 % 200 0
% T4:16 % 200 0
% T4:17 % 200 0
% T4:18 % 200 0
DATA C5
% .PRE .ACC %
% C5:0 % 25 0
DATA N7
% N7:10 % 0 0 0 0 31200 31200 0 0 0 0
DATA N14
% N14:10 % 960 960 3 16191 0 0 0 0 0 0
% N14:20 % 0 5 300 0 4 300 0 0 0 0
